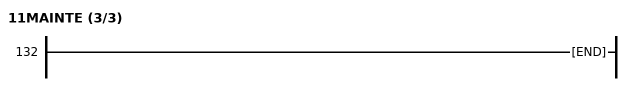
[picture p48: ladder of 11MAINTE, rungs at steps 132 to 132]
132   END
END_PROGRAM

PROGRAM 12ALARM1
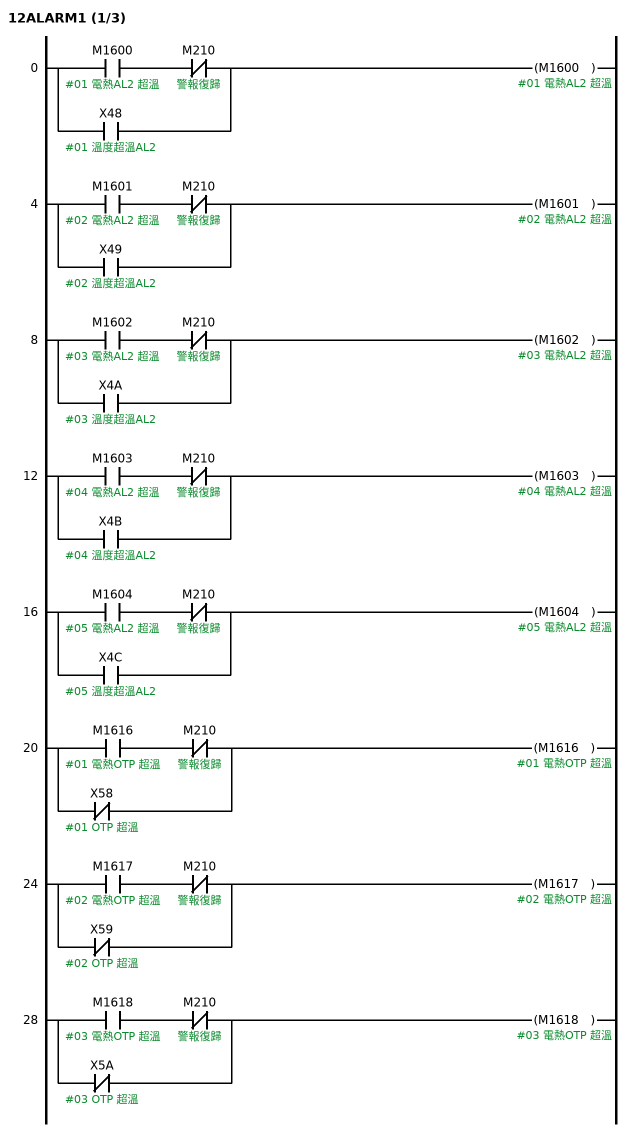
0     LD      M1600  ; #01 電熱AL2 超溫
      ANI     M210  ; 警報復歸
      OR      X48  ; #01 溫度超溫AL2
      OUT     M1600  ; #01 電熱AL2 超溫
4     LD      M1601  ; #02 電熱AL2 超溫
      ANI     M210  ; 警報復歸
      OR      X49  ; #02 溫度超溫AL2
      OUT     M1601  ; #02 電熱AL2 超溫
8     LD      M1602  ; #03 電熱AL2 超溫
      ANI     M210  ; 警報復歸
      OR      X4A  ; #03 溫度超溫AL2
      OUT     M1602  ; #03 電熱AL2 超溫
12    LD      M1603  ; #04 電熱AL2 超溫
      ANI     M210  ; 警報復歸
      OR      X4B  ; #04 溫度超溫AL2
      OUT     M1603  ; #04 電熱AL2 超溫
16    LD      M1604  ; #05 電熱AL2 超溫
      ANI     M210  ; 警報復歸
      OR      X4C  ; #05 溫度超溫AL2
      OUT     M1604  ; #05 電熱AL2 超溫
20    LD      M1616  ; #01 電熱OTP 超溫
      ANI     M210  ; 警報復歸
      ORI     X58  ; #01 OTP 超溫
      OUT     M1616  ; #01 電熱OTP 超溫
24    LD      M1617  ; #02 電熱OTP 超溫
      ANI     M210  ; 警報復歸
      ORI     X59  ; #02 OTP 超溫
      OUT     M1617  ; #02 電熱OTP 超溫
28    LD      M1618  ; #03 電熱OTP 超溫
      ANI     M210  ; 警報復歸
      ORI     X5A  ; #03 OTP 超溫
      OUT     M1618  ; #03 電熱OTP 超溫
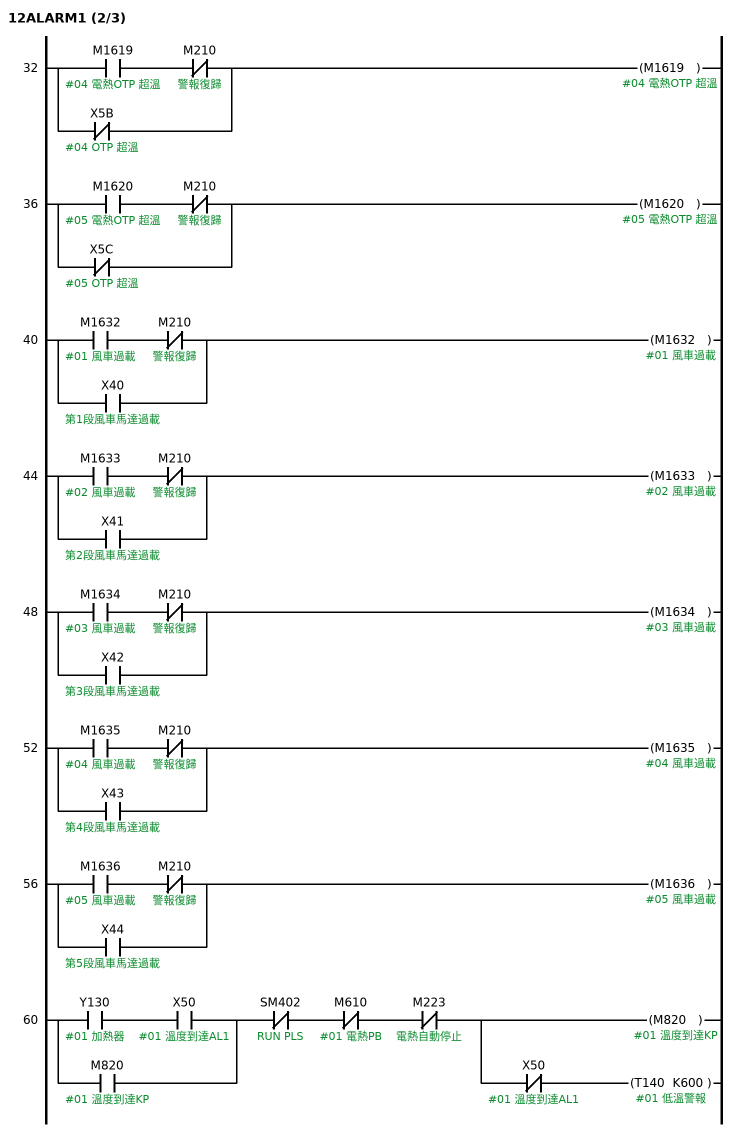
32    LD      M1619  ; #04 電熱OTP 超溫
      ANI     M210  ; 警報復歸
      ORI     X5B  ; #04 OTP 超溫
      OUT     M1619  ; #04 電熱OTP 超溫
36    LD      M1620  ; #05 電熱OTP 超溫
      ANI     M210  ; 警報復歸
      ORI     X5C  ; #05 OTP 超溫
      OUT     M1620  ; #05 電熱OTP 超溫
40    LD      M1632  ; #01 風車過載
      ANI     M210  ; 警報復歸
      OR      X40  ; 第1段風車馬達過載
      OUT     M1632  ; #01 風車過載
44    LD      M1633  ; #02 風車過載
      ANI     M210  ; 警報復歸
      OR      X41  ; 第2段風車馬達過載
      OUT     M1633  ; #02 風車過載
48    LD      M1634  ; #03 風車過載
      ANI     M210  ; 警報復歸
      OR      X42  ; 第3段風車馬達過載
      OUT     M1634  ; #03 風車過載
52    LD      M1635  ; #04 風車過載
      ANI     M210  ; 警報復歸
      OR      X43  ; 第4段風車馬達過載
      OUT     M1635  ; #04 風車過載
56    LD      M1636  ; #05 風車過載
      ANI     M210  ; 警報復歸
      OR      X44  ; 第5段風車馬達過載
      OUT     M1636  ; #05 風車過載
60    LD      Y130  ; #01 加熱器
      AND     X50  ; #01 溫度到達AL1
      OR      M820  ; #01 溫度到達KP
      ANI     SM402  ; RUN PLS
      ANI     M610  ; #01 電熱PB
      ANI     M223  ; 電熱自動停止
      OUT     M820  ; #01 溫度到達KP
      ANI     X50  ; #01 溫度到達AL1
      OUT     T140 K600  ; #01 低溫警報
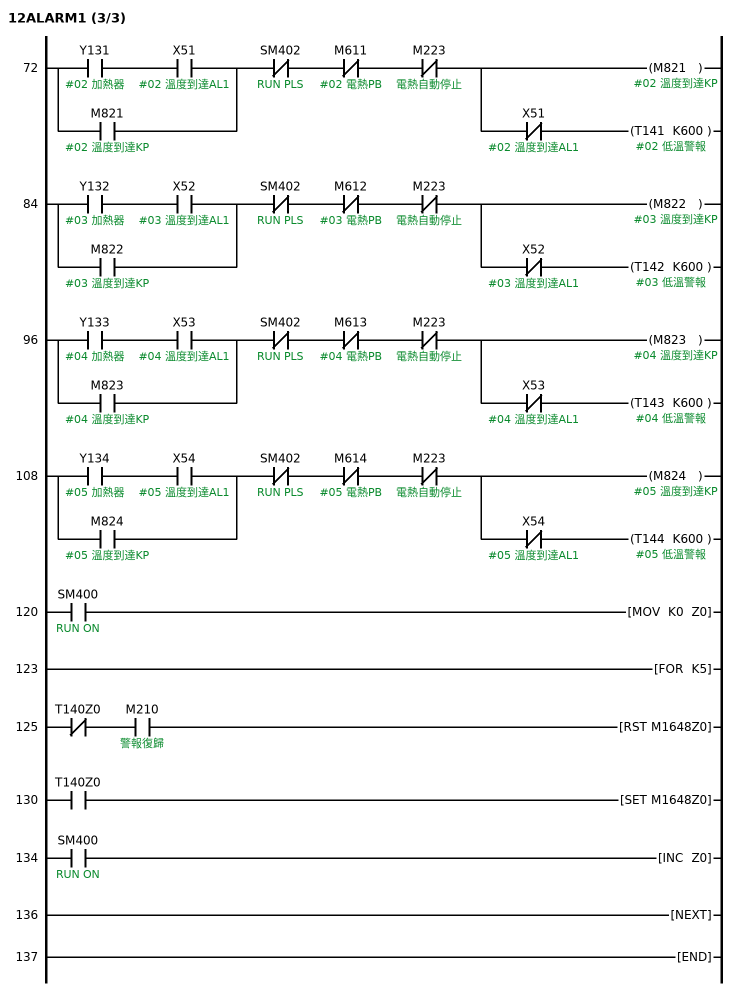
72    LD      Y131  ; #02 加熱器
      AND     X51  ; #02 溫度到達AL1
      OR      M821  ; #02 溫度到達KP
      ANI     SM402  ; RUN PLS
      ANI     M611  ; #02 電熱PB
      ANI     M223  ; 電熱自動停止
      OUT     M821  ; #02 溫度到達KP
      ANI     X51  ; #02 溫度到達AL1
      OUT     T141 K600  ; #02 低溫警報
84    LD      Y132  ; #03 加熱器
      AND     X52  ; #03 溫度到達AL1
      OR      M822  ; #03 溫度到達KP
      ANI     SM402  ; RUN PLS
      ANI     M612  ; #03 電熱PB
      ANI     M223  ; 電熱自動停止
      OUT     M822  ; #03 溫度到達KP
      ANI     X52  ; #03 溫度到達AL1
      OUT     T142 K600  ; #03 低溫警報
96    LD      Y133  ; #04 加熱器
      AND     X53  ; #04 溫度到達AL1
      OR      M823  ; #04 溫度到達KP
      ANI     SM402  ; RUN PLS
      ANI     M613  ; #04 電熱PB
      ANI     M223  ; 電熱自動停止
      OUT     M823  ; #04 溫度到達KP
      ANI     X53  ; #04 溫度到達AL1
      OUT     T143 K600  ; #04 低溫警報
108   LD      Y134  ; #05 加熱器
      AND     X54  ; #05 溫度到達AL1
      OR      M824  ; #05 溫度到達KP
      ANI     SM402  ; RUN PLS
      ANI     M614  ; #05 電熱PB
      ANI     M223  ; 電熱自動停止
      OUT     M824  ; #05 溫度到達KP
      ANI     X54  ; #05 溫度到達AL1
      OUT     T144 K600  ; #05 低溫警報
120   LD      SM400  ; RUN ON
      MOV     K0 Z0
123   FOR     K5
125   LDI     T140Z0
      AND     M210  ; 警報復歸
      RST     M1648Z0
130   LD      T140Z0
      SET     M1648Z0
134   LD      SM400  ; RUN ON
      INC     Z0
136   NEXT
137   END
END_PROGRAM

PROGRAM 13ALARM2
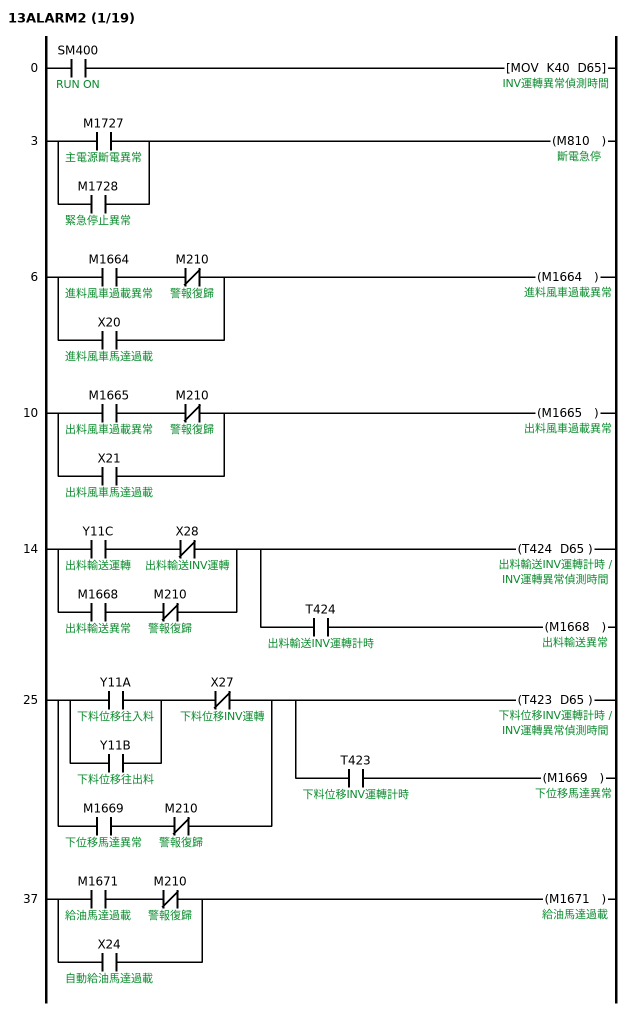
0     LD      SM400  ; RUN ON
      MOV     K40 D65  ; INV運轉異常偵測時間
3     LD      M1727  ; 主電源斷電異常
      OR      M1728  ; 緊急停止異常
      OUT     M810  ; 斷電急停
6     LD      M1664  ; 進料風車過載異常
      ANI     M210  ; 警報復歸
      OR      X20  ; 進料風車馬達過載
      OUT     M1664  ; 進料風車過載異常
10    LD      M1665  ; 出料風車過載異常
      ANI     M210  ; 警報復歸
      OR      X21  ; 出料風車馬達過載
      OUT     M1665  ; 出料風車過載異常
14    LD      Y11C  ; 出料輸送運轉
      ANI     X28  ; 出料輸送INV運轉
      LD      M1668  ; 出料輸送異常
      ANI     M210  ; 警報復歸
      ORB
      OUT     T424 D65  ; 出料輸送INV運轉計時 / INV運轉異常偵測時間
      AND     T424  ; 出料輸送INV運轉計時
      OUT     M1668  ; 出料輸送異常
25    LD      Y11A  ; 下料位移往入料
      OR      Y11B  ; 下料位移往出料
      ANI     X27  ; 下料位移INV運轉
      LD      M1669  ; 下位移馬達異常
      ANI     M210  ; 警報復歸
      ORB
      OUT     T423 D65  ; 下料位移INV運轉計時 / INV運轉異常偵測時間
      AND     T423  ; 下料位移INV運轉計時
      OUT     M1669  ; 下位移馬達異常
37    LD      M1671  ; 給油馬達過載
      ANI     M210  ; 警報復歸
      OR      X24  ; 自動給油馬達過載
      OUT     M1671  ; 給油馬達過載
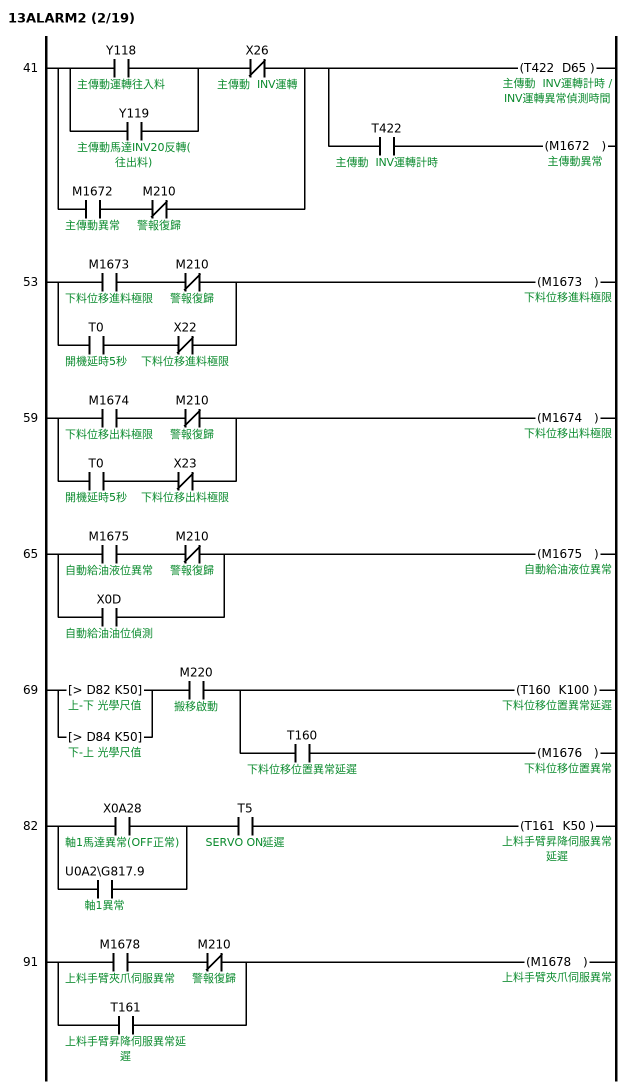
41    LD      Y118  ; 主傳動運轉往入料
      OR      Y119  ; 主傳動馬達INV20反轉(往出料)
      ANI     X26  ; 主傳動  INV運轉
      LD      M1672  ; 主傳動異常
      ANI     M210  ; 警報復歸
      ORB
      OUT     T422 D65  ; 主傳動  INV運轉計時 / INV運轉異常偵測時間
      AND     T422  ; 主傳動  INV運轉計時
      OUT     M1672  ; 主傳動異常
53    LD      M1673  ; 下料位移進料極限
      ANI     M210  ; 警報復歸
      LD      T0  ; 開機延時5秒
      ANI     X22  ; 下料位移進料極限
      ORB
      OUT     M1673  ; 下料位移進料極限
59    LD      M1674  ; 下料位移出料極限
      ANI     M210  ; 警報復歸
      LD      T0  ; 開機延時5秒
      ANI     X23  ; 下料位移出料極限
      ORB
      OUT     M1674  ; 下料位移出料極限
65    LD      M1675  ; 自動給油液位異常
      ANI     M210  ; 警報復歸
      OR      X0D  ; 自動給油油位偵測
      OUT     M1675  ; 自動給油液位異常
69    LD>     D82 K50  ; 上-下 光學尺值
      OR>     D84 K50  ; 下-上 光學尺值
      AND     M220  ; 搬移啟動
      OUT     T160 K100  ; 下料位移位置異常延遲
      AND     T160  ; 下料位移位置異常延遲
      OUT     M1676  ; 下料位移位置異常
82    LD      X0A28  ; 軸1馬達異常(OFF正常)
      OR      U0A2\G817.9  ; 軸1異常
      AND     T5  ; SERVO ON延遲
      OUT     T161 K50  ; 上料手臂昇降伺服異常延遲
91    LD      M1678  ; 上料手臂夾爪伺服異常
      ANI     M210  ; 警報復歸
      OR      T161  ; 上料手臂昇降伺服異常延遲
      OUT     M1678  ; 上料手臂夾爪伺服異常
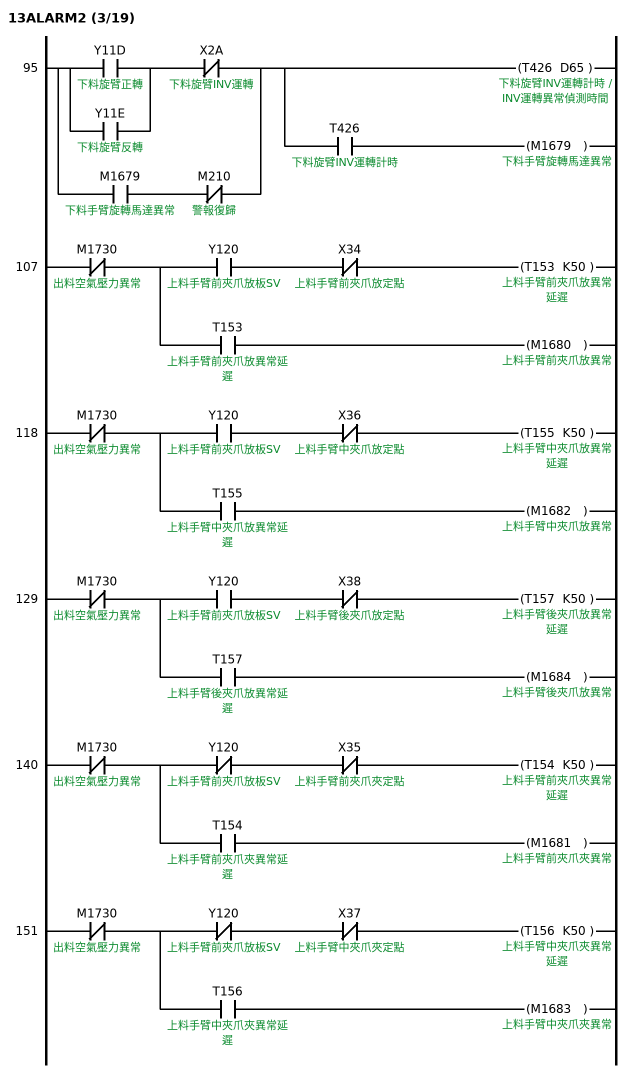
95    LD      Y11D  ; 下料旋臂正轉
      OR      Y11E  ; 下料旋臂反轉
      ANI     X2A  ; 下料旋臂INV運轉
      LD      M1679  ; 下料手臂旋轉馬達異常
      ANI     M210  ; 警報復歸
      ORB
      OUT     T426 D65  ; 下料旋臂INV運轉計時 / INV運轉異常偵測時間
      AND     T426  ; 下料旋臂INV運轉計時
      OUT     M1679  ; 下料手臂旋轉馬達異常
107   LDI     M1730  ; 出料空氣壓力異常
      MPS
      AND     Y120  ; 上料手臂前夾爪放板SV
      ANI     X34  ; 上料手臂前夾爪放定點
      OUT     T153 K50  ; 上料手臂前夾爪放異常延遲
      MPP
      AND     T153  ; 上料手臂前夾爪放異常延遲
      OUT     M1680  ; 上料手臂前夾爪放異常
118   LDI     M1730  ; 出料空氣壓力異常
      MPS
      AND     Y120  ; 上料手臂前夾爪放板SV
      ANI     X36  ; 上料手臂中夾爪放定點
      OUT     T155 K50  ; 上料手臂中夾爪放異常延遲
      MPP
      AND     T155  ; 上料手臂中夾爪放異常延遲
      OUT     M1682  ; 上料手臂中夾爪放異常
129   LDI     M1730  ; 出料空氣壓力異常
      MPS
      AND     Y120  ; 上料手臂前夾爪放板SV
      ANI     X38  ; 上料手臂後夾爪放定點
      OUT     T157 K50  ; 上料手臂後夾爪放異常延遲
      MPP
      AND     T157  ; 上料手臂後夾爪放異常延遲
      OUT     M1684  ; 上料手臂後夾爪放異常
140   LDI     M1730  ; 出料空氣壓力異常
      MPS
      ANI     Y120  ; 上料手臂前夾爪放板SV
      ANI     X35  ; 上料手臂前夾爪夾定點
      OUT     T154 K50  ; 上料手臂前夾爪夾異常延遲
      MPP
      AND     T154  ; 上料手臂前夾爪夾異常延遲
      OUT     M1681  ; 上料手臂前夾爪夾異常
151   LDI     M1730  ; 出料空氣壓力異常
      MPS
      ANI     Y120  ; 上料手臂前夾爪放板SV
      ANI     X37  ; 上料手臂中夾爪夾定點
      OUT     T156 K50  ; 上料手臂中夾爪夾異常延遲
      MPP
      AND     T156  ; 上料手臂中夾爪夾異常延遲
      OUT     M1683  ; 上料手臂中夾爪夾異常
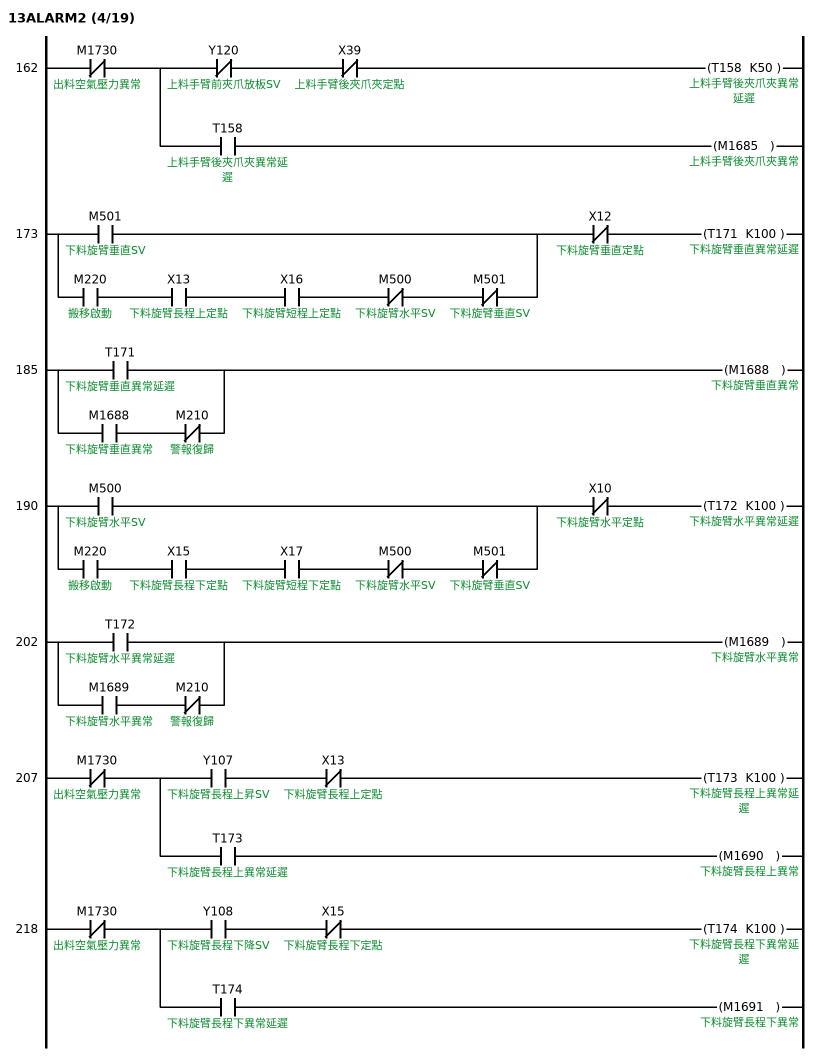
162   LDI     M1730  ; 出料空氣壓力異常
      MPS
      ANI     Y120  ; 上料手臂前夾爪放板SV
      ANI     X39  ; 上料手臂後夾爪夾定點
      OUT     T158 K50  ; 上料手臂後夾爪夾異常延遲
      MPP
      AND     T158  ; 上料手臂後夾爪夾異常延遲
      OUT     M1685  ; 上料手臂後夾爪夾異常
173   LD      M501  ; 下料旋臂垂直SV
      LD      M220  ; 搬移啟動
      AND     X13  ; 下料旋臂長程上定點
      AND     X16  ; 下料旋臂短程上定點
      ANI     M500  ; 下料旋臂水平SV
      ANI     M501  ; 下料旋臂垂直SV
      ORB
      ANI     X12  ; 下料旋臂垂直定點
      OUT     T171 K100  ; 下料旋臂垂直異常延遲
185   LD      T171  ; 下料旋臂垂直異常延遲
      LD      M1688  ; 下料旋臂垂直異常
      ANI     M210  ; 警報復歸
      ORB
      OUT     M1688  ; 下料旋臂垂直異常
190   LD      M500  ; 下料旋臂水平SV
      LD      M220  ; 搬移啟動
      AND     X15  ; 下料旋臂長程下定點
      AND     X17  ; 下料旋臂短程下定點
      ANI     M500  ; 下料旋臂水平SV
      ANI     M501  ; 下料旋臂垂直SV
      ORB
      ANI     X10  ; 下料旋臂水平定點
      OUT     T172 K100  ; 下料旋臂水平異常延遲
202   LD      T172  ; 下料旋臂水平異常延遲
      LD      M1689  ; 下料旋臂水平異常
      ANI     M210  ; 警報復歸
      ORB
      OUT     M1689  ; 下料旋臂水平異常
207   LDI     M1730  ; 出料空氣壓力異常
      MPS
      AND     Y107  ; 下料旋臂長程上昇SV
      ANI     X13  ; 下料旋臂長程上定點
      OUT     T173 K100  ; 下料旋臂長程上異常延遲
      MPP
      AND     T173  ; 下料旋臂長程上異常延遲
      OUT     M1690  ; 下料旋臂長程上異常
218   LDI     M1730  ; 出料空氣壓力異常
      MPS
      AND     Y108  ; 下料旋臂長程下降SV
      ANI     X15  ; 下料旋臂長程下定點
      OUT     T174 K100  ; 下料旋臂長程下異常延遲
      MPP
      AND     T174  ; 下料旋臂長程下異常延遲
      OUT     M1691  ; 下料旋臂長程下異常
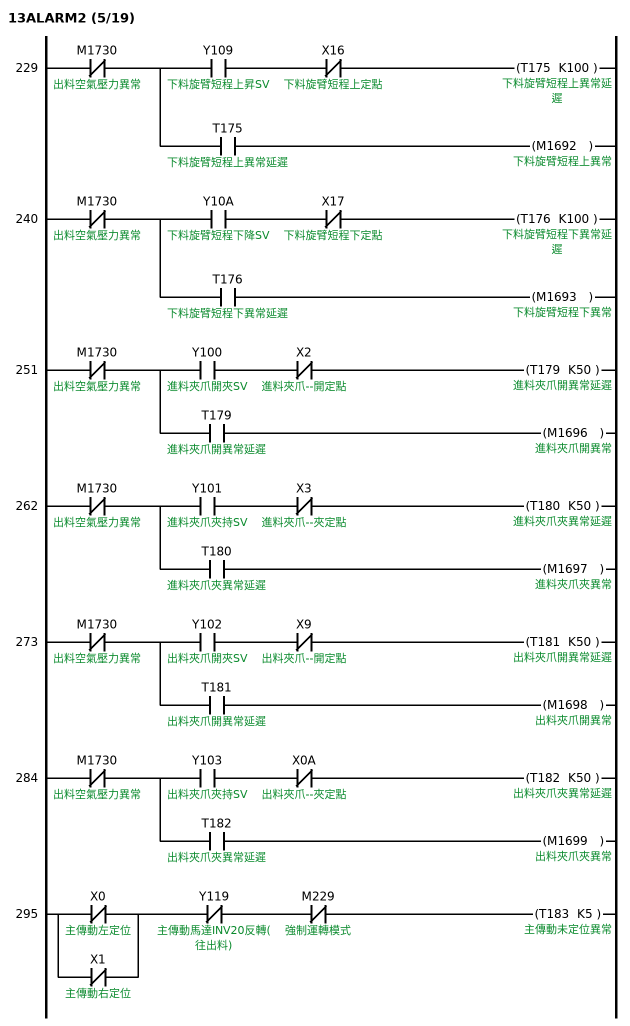
229   LDI     M1730  ; 出料空氣壓力異常
      MPS
      AND     Y109  ; 下料旋臂短程上昇SV
      ANI     X16  ; 下料旋臂短程上定點
      OUT     T175 K100  ; 下料旋臂短程上異常延遲
      MPP
      AND     T175  ; 下料旋臂短程上異常延遲
      OUT     M1692  ; 下料旋臂短程上異常
240   LDI     M1730  ; 出料空氣壓力異常
      MPS
      AND     Y10A  ; 下料旋臂短程下降SV
      ANI     X17  ; 下料旋臂短程下定點
      OUT     T176 K100  ; 下料旋臂短程下異常延遲
      MPP
      AND     T176  ; 下料旋臂短程下異常延遲
      OUT     M1693  ; 下料旋臂短程下異常
251   LDI     M1730  ; 出料空氣壓力異常
      MPS
      AND     Y100  ; 進料夾爪開夾SV
      ANI     X2  ; 進料夾爪--開定點
      OUT     T179 K50  ; 進料夾爪開異常延遲
      MPP
      AND     T179  ; 進料夾爪開異常延遲
      OUT     M1696  ; 進料夾爪開異常
262   LDI     M1730  ; 出料空氣壓力異常
      MPS
      AND     Y101  ; 進料夾爪夾持SV
      ANI     X3  ; 進料夾爪--夾定點
      OUT     T180 K50  ; 進料夾爪夾異常延遲
      MPP
      AND     T180  ; 進料夾爪夾異常延遲
      OUT     M1697  ; 進料夾爪夾異常
273   LDI     M1730  ; 出料空氣壓力異常
      MPS
      AND     Y102  ; 出料夾爪開夾SV
      ANI     X9  ; 出料夾爪--開定點
      OUT     T181 K50  ; 出料夾爪開異常延遲
      MPP
      AND     T181  ; 出料夾爪開異常延遲
      OUT     M1698  ; 出料夾爪開異常
284   LDI     M1730  ; 出料空氣壓力異常
      MPS
      AND     Y103  ; 出料夾爪夾持SV
      ANI     X0A  ; 出料夾爪--夾定點
      OUT     T182 K50  ; 出料夾爪夾異常延遲
      MPP
      AND     T182  ; 出料夾爪夾異常延遲
      OUT     M1699  ; 出料夾爪夾異常
295   LDI     X0  ; 主傳動左定位
      ORI     X1  ; 主傳動右定位
      ANI     Y119  ; 主傳動馬達INV20反轉(往出料)
      ANI     M229  ; 強制運轉模式
      OUT     T183 K5  ; 主傳動未定位異常
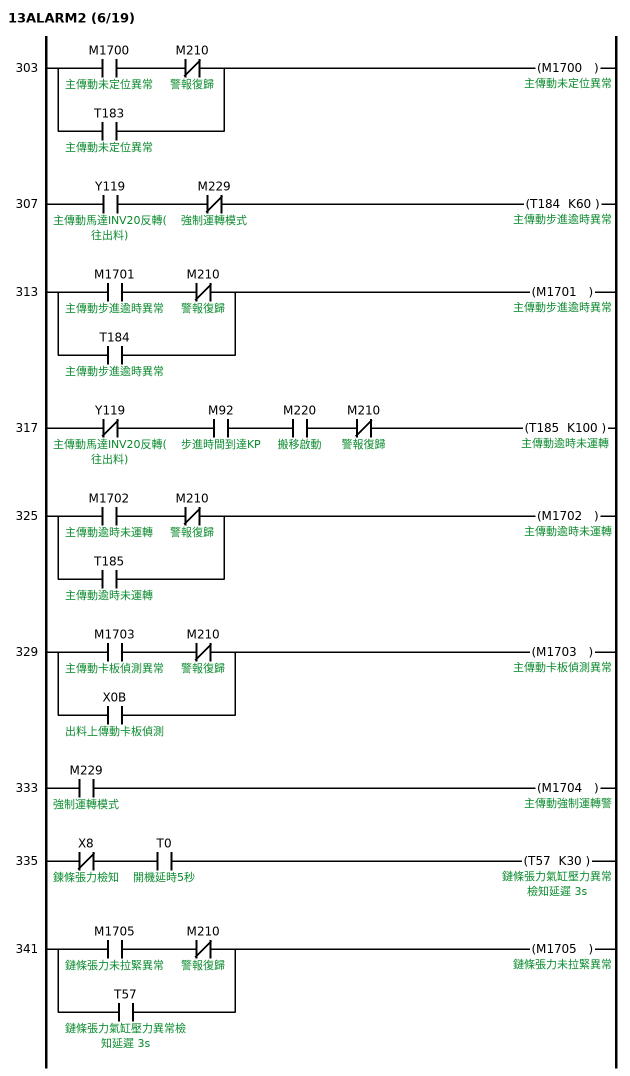
303   LD      M1700  ; 主傳動未定位異常
      ANI     M210  ; 警報復歸
      OR      T183  ; 主傳動未定位異常
      OUT     M1700  ; 主傳動未定位異常
307   LD      Y119  ; 主傳動馬達INV20反轉(往出料)
      ANI     M229  ; 強制運轉模式
      OUT     T184 K60  ; 主傳動步進逾時異常
313   LD      M1701  ; 主傳動步進逾時異常
      ANI     M210  ; 警報復歸
      OR      T184  ; 主傳動步進逾時異常
      OUT     M1701  ; 主傳動步進逾時異常
317   LDI     Y119  ; 主傳動馬達INV20反轉(往出料)
      AND     M92  ; 步進時間到達KP
      AND     M220  ; 搬移啟動
      ANI     M210  ; 警報復歸
      OUT     T185 K100  ; 主傳動逾時未運轉
325   LD      M1702  ; 主傳動逾時未運轉
      ANI     M210  ; 警報復歸
      OR      T185  ; 主傳動逾時未運轉
      OUT     M1702  ; 主傳動逾時未運轉
329   LD      M1703  ; 主傳動卡板偵測異常
      ANI     M210  ; 警報復歸
      OR      X0B  ; 出料上傳動卡板偵測
      OUT     M1703  ; 主傳動卡板偵測異常
333   LD      M229  ; 強制運轉模式
      OUT     M1704  ; 主傳動強制運轉警
335   LDI     X8  ; 鍊條張力檢知
      AND     T0  ; 開機延時5秒
      OUT     T57 K30  ; 鏈條張力氣缸壓力異常檢知延遲 3s
341   LD      M1705  ; 鏈條張力未拉緊異常
      ANI     M210  ; 警報復歸
      OR      T57  ; 鏈條張力氣缸壓力異常檢知延遲 3s
      OUT     M1705  ; 鏈條張力未拉緊異常
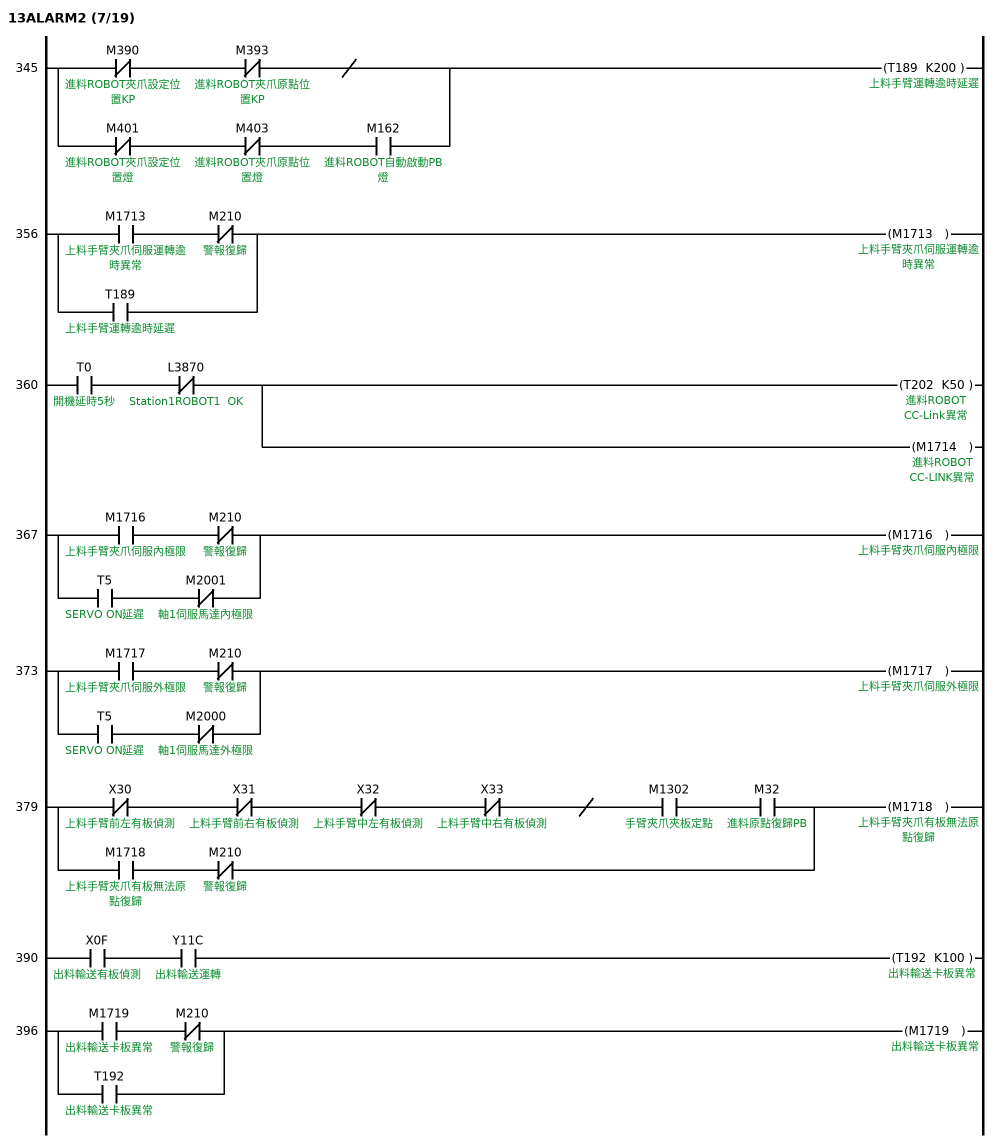
345   LDI     M390  ; 進料ROBOT夾爪設定位置KP
      ANI     M393  ; 進料ROBOT夾爪原點位置KP
      INV
      LDI     M401  ; 進料ROBOT夾爪設定位置燈
      ANI     M403  ; 進料ROBOT夾爪原點位置燈
      AND     M162  ; 進料ROBOT自動啟動PB燈
      ORB
      OUT     T189 K200  ; 上料手臂運轉逾時延遲
356   LD      M1713  ; 上料手臂夾爪伺服運轉逾時異常
      ANI     M210  ; 警報復歸
      OR      T189  ; 上料手臂運轉逾時延遲
      OUT     M1713  ; 上料手臂夾爪伺服運轉逾時異常
360   LD      T0  ; 開機延時5秒
      ANI     L3870  ; Station1ROBOT1  OK
      OUT     T202 K50  ; 進料ROBOT CC-Link異常
      OUT     M1714  ; 進料ROBOT CC-LINK異常
367   LD      M1716  ; 上料手臂夾爪伺服內極限
      ANI     M210  ; 警報復歸
      LD      T5  ; SERVO ON延遲
      ANI     M2001  ; 軸1伺服馬達內極限
      ORB
      OUT     M1716  ; 上料手臂夾爪伺服內極限
373   LD      M1717  ; 上料手臂夾爪伺服外極限
      ANI     M210  ; 警報復歸
      LD      T5  ; SERVO ON延遲
      ANI     M2000  ; 軸1伺服馬達外極限
      ORB
      OUT     M1717  ; 上料手臂夾爪伺服外極限
379   LDI     X30  ; 上料手臂前左有板偵測
      ANI     X31  ; 上料手臂前右有板偵測
      ANI     X32  ; 上料手臂中左有板偵測
      ANI     X33  ; 上料手臂中右有板偵測
      INV
      AND     M1302  ; 手臂夾爪夾板定點
      AND     M32  ; 進料原點復歸PB
      LD      M1718  ; 上料手臂夾爪有板無法原點復歸
      ANI     M210  ; 警報復歸
      ORB
      OUT     M1718  ; 上料手臂夾爪有板無法原點復歸
390   LD      X0F  ; 出料輸送有板偵測
      AND     Y11C  ; 出料輸送運轉
      OUT     T192 K100  ; 出料輸送卡板異常
396   LD      M1719  ; 出料輸送卡板異常
      ANI     M210  ; 警報復歸
      OR      T192  ; 出料輸送卡板異常
      OUT     M1719  ; 出料輸送卡板異常
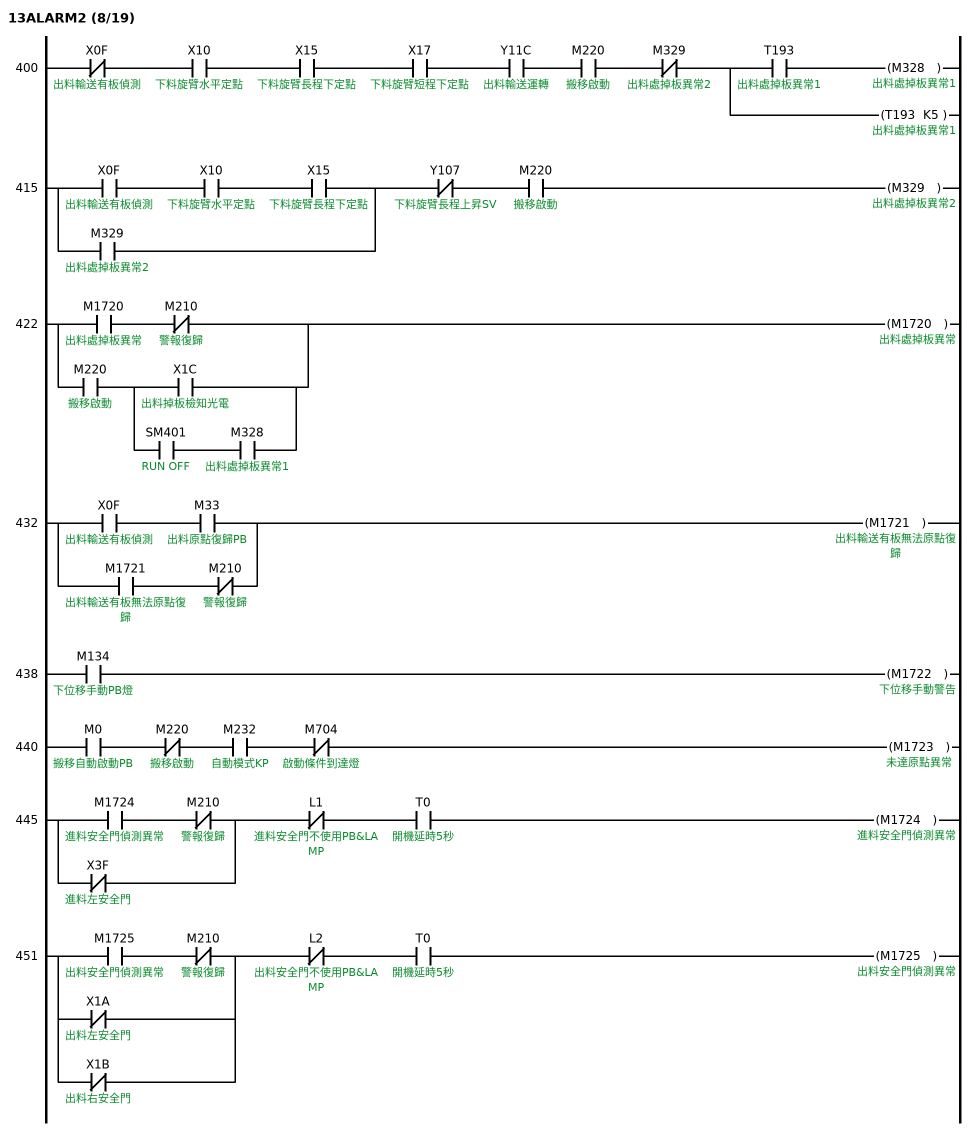
400   LDI     X0F  ; 出料輸送有板偵測
      AND     X10  ; 下料旋臂水平定點
      AND     X15  ; 下料旋臂長程下定點
      AND     X17  ; 下料旋臂短程下定點
      AND     Y11C  ; 出料輸送運轉
      AND     M220  ; 搬移啟動
      ANI     M329  ; 出料處掉板異常2
      MPS
      AND     T193  ; 出料處掉板異常1
      OUT     M328  ; 出料處掉板異常1
      MPP
      OUT     T193 K5  ; 出料處掉板異常1
415   LD      X0F  ; 出料輸送有板偵測
      AND     X10  ; 下料旋臂水平定點
      AND     X15  ; 下料旋臂長程下定點
      OR      M329  ; 出料處掉板異常2
      ANI     Y107  ; 下料旋臂長程上昇SV
      AND     M220  ; 搬移啟動
      OUT     M329  ; 出料處掉板異常2
422   LD      M1720  ; 出料處掉板異常
      ANI     M210  ; 警報復歸
      LD      M220  ; 搬移啟動
      LD      X1C  ; 出料掉板檢知光電
      LD      SM401  ; RUN OFF
      AND     M328  ; 出料處掉板異常1
      ORB
      ANB
      ORB
      OUT     M1720  ; 出料處掉板異常
432   LD      X0F  ; 出料輸送有板偵測
      AND     M33  ; 出料原點復歸PB
      LD      M1721  ; 出料輸送有板無法原點復歸
      ANI     M210  ; 警報復歸
      ORB
      OUT     M1721  ; 出料輸送有板無法原點復歸
438   LD      M134  ; 下位移手動PB燈
      OUT     M1722  ; 下位移手動警告
440   LD      M0  ; 搬移自動啟動PB
      ANI     M220  ; 搬移啟動
      AND     M232  ; 自動模式KP
      ANI     M704  ; 啟動條件到達燈
      OUT     M1723  ; 未達原點異常
445   LD      M1724  ; 進料安全門偵測異常
      ANI     M210  ; 警報復歸
      ORI     X3F  ; 進料左安全門
      ANI     L1  ; 進料安全門不使用PB&LAMP
      AND     T0  ; 開機延時5秒
      OUT     M1724  ; 進料安全門偵測異常
451   LD      M1725  ; 出料安全門偵測異常
      ANI     M210  ; 警報復歸
      ORI     X1A  ; 出料左安全門
      ORI     X1B  ; 出料右安全門
      ANI     L2  ; 出料安全門不使用PB&LAMP
      AND     T0  ; 開機延時5秒
      OUT     M1725  ; 出料安全門偵測異常
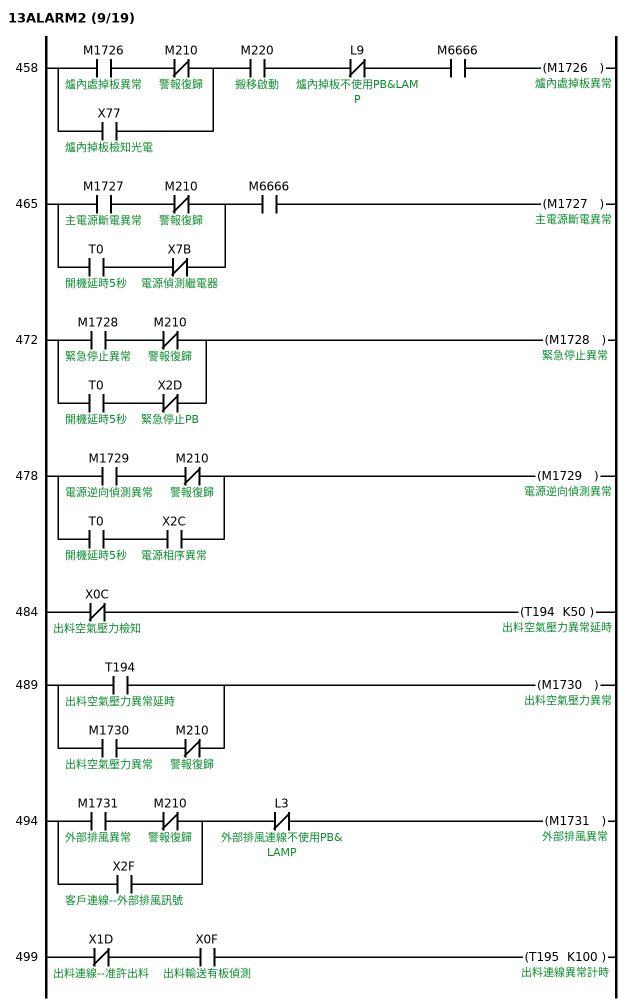
458   LD      M1726  ; 爐內處掉板異常
      ANI     M210  ; 警報復歸
      OR      X77  ; 爐內掉板檢知光電
      AND     M220  ; 搬移啟動
      ANI     L9  ; 爐內掉板不使用PB&LAMP
      AND     M6666
      OUT     M1726  ; 爐內處掉板異常
465   LD      M1727  ; 主電源斷電異常
      ANI     M210  ; 警報復歸
      LD      T0  ; 開機延時5秒
      ANI     X7B  ; 電源偵測繼電器
      ORB
      AND     M6666
      OUT     M1727  ; 主電源斷電異常
472   LD      M1728  ; 緊急停止異常
      ANI     M210  ; 警報復歸
      LD      T0  ; 開機延時5秒
      ANI     X2D  ; 緊急停止PB
      ORB
      OUT     M1728  ; 緊急停止異常
478   LD      M1729  ; 電源逆向偵測異常
      ANI     M210  ; 警報復歸
      LD      T0  ; 開機延時5秒
      AND     X2C  ; 電源相序異常
      ORB
      OUT     M1729  ; 電源逆向偵測異常
484   LDI     X0C  ; 出料空氣壓力檢知
      OUT     T194 K50  ; 出料空氣壓力異常延時
489   LD      T194  ; 出料空氣壓力異常延時
      LD      M1730  ; 出料空氣壓力異常
      ANI     M210  ; 警報復歸
      ORB
      OUT     M1730  ; 出料空氣壓力異常
494   LD      M1731  ; 外部排風異常
      ANI     M210  ; 警報復歸
      OR      X2F  ; 客戶連線--外部排風訊號
      ANI     L3  ; 外部排風連線不使用PB&LAMP
      OUT     M1731  ; 外部排風異常
499   LDI     X1D  ; 出料連線--准許出料
      AND     X0F  ; 出料輸送有板偵測
      OUT     T195 K100  ; 出料連線異常計時
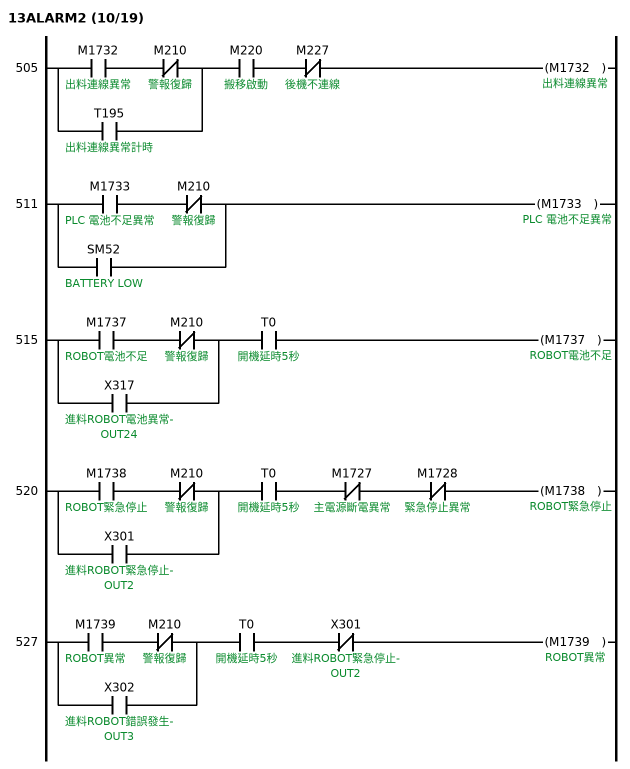
505   LD      M1732  ; 出料連線異常
      ANI     M210  ; 警報復歸
      OR      T195  ; 出料連線異常計時
      AND     M220  ; 搬移啟動
      ANI     M227  ; 後機不連線
      OUT     M1732  ; 出料連線異常
511   LD      M1733  ; PLC 電池不足異常
      ANI     M210  ; 警報復歸
      OR      SM52  ; BATTERY LOW
      OUT     M1733  ; PLC 電池不足異常
515   LD      M1737  ; ROBOT電池不足
      ANI     M210  ; 警報復歸
      OR      X317  ; 進料ROBOT電池異常-OUT24
      AND     T0  ; 開機延時5秒
      OUT     M1737  ; ROBOT電池不足
520   LD      M1738  ; ROBOT緊急停止
      ANI     M210  ; 警報復歸
      OR      X301  ; 進料ROBOT緊急停止-OUT2
      AND     T0  ; 開機延時5秒
      ANI     M1727  ; 主電源斷電異常
      ANI     M1728  ; 緊急停止異常
      OUT     M1738  ; ROBOT緊急停止
527   LD      M1739  ; ROBOT異常
      ANI     M210  ; 警報復歸
      OR      X302  ; 進料ROBOT錯誤發生-OUT3
      AND     T0  ; 開機延時5秒
      ANI     X301  ; 進料ROBOT緊急停止-OUT2
      OUT     M1739  ; ROBOT異常
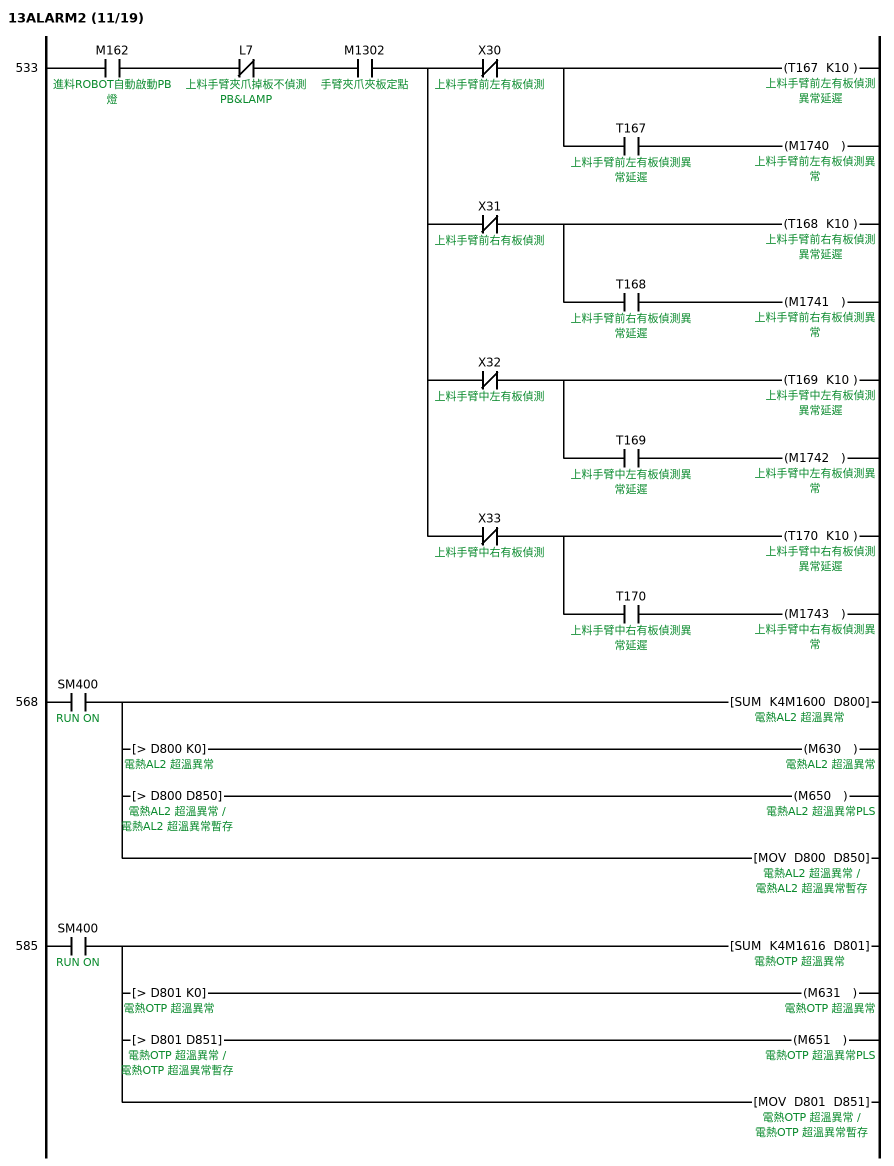
533   LD      M162  ; 進料ROBOT自動啟動PB燈
      ANI     L7  ; 上料手臂夾爪掉板不偵測PB&LAMP
      AND     M1302  ; 手臂夾爪夾板定點
      MPS
      ANI     X30  ; 上料手臂前左有板偵測
      OUT     T167 K10  ; 上料手臂前左有板偵測異常延遲
      AND     T167  ; 上料手臂前左有板偵測異常延遲
      OUT     M1740  ; 上料手臂前左有板偵測異常
      MRD
      ANI     X31  ; 上料手臂前右有板偵測
      OUT     T168 K10  ; 上料手臂前右有板偵測異常延遲
      AND     T168  ; 上料手臂前右有板偵測異常延遲
      OUT     M1741  ; 上料手臂前右有板偵測異常
      MRD
      ANI     X32  ; 上料手臂中左有板偵測
      OUT     T169 K10  ; 上料手臂中左有板偵測異常延遲
      AND     T169  ; 上料手臂中左有板偵測異常延遲
      OUT     M1742  ; 上料手臂中左有板偵測異常
      MPP
      ANI     X33  ; 上料手臂中右有板偵測
      OUT     T170 K10  ; 上料手臂中右有板偵測異常延遲
      AND     T170  ; 上料手臂中右有板偵測異常延遲
      OUT     M1743  ; 上料手臂中右有板偵測異常
568   LD      SM400  ; RUN ON
      SUM     K4M1600 D800  ; #01 電熱AL2 超溫 / 電熱AL2 超溫異常
      MPS
      AND>    D800 K0  ; 電熱AL2 超溫異常
      OUT     M630  ; 電熱AL2 超溫異常
      MRD
      AND>    D800 D850  ; 電熱AL2 超溫異常 / 電熱AL2 超溫異常暫存
      OUT     M650  ; 電熱AL2 超溫異常PLS
      MPP
      MOV     D800 D850
585   LD      SM400  ; RUN ON
      SUM     K4M1616 D801  ; #01 電熱OTP 超溫 / 電熱OTP 超溫異常
      MPS
      AND>    D801 K0  ; 電熱OTP 超溫異常
      OUT     M631  ; 電熱OTP 超溫異常
      MRD
      AND>    D801 D851  ; 電熱OTP 超溫異常 / 電熱OTP 超溫異常暫存
      OUT     M651  ; 電熱OTP 超溫異常PLS
      MPP
      MOV     D801 D851
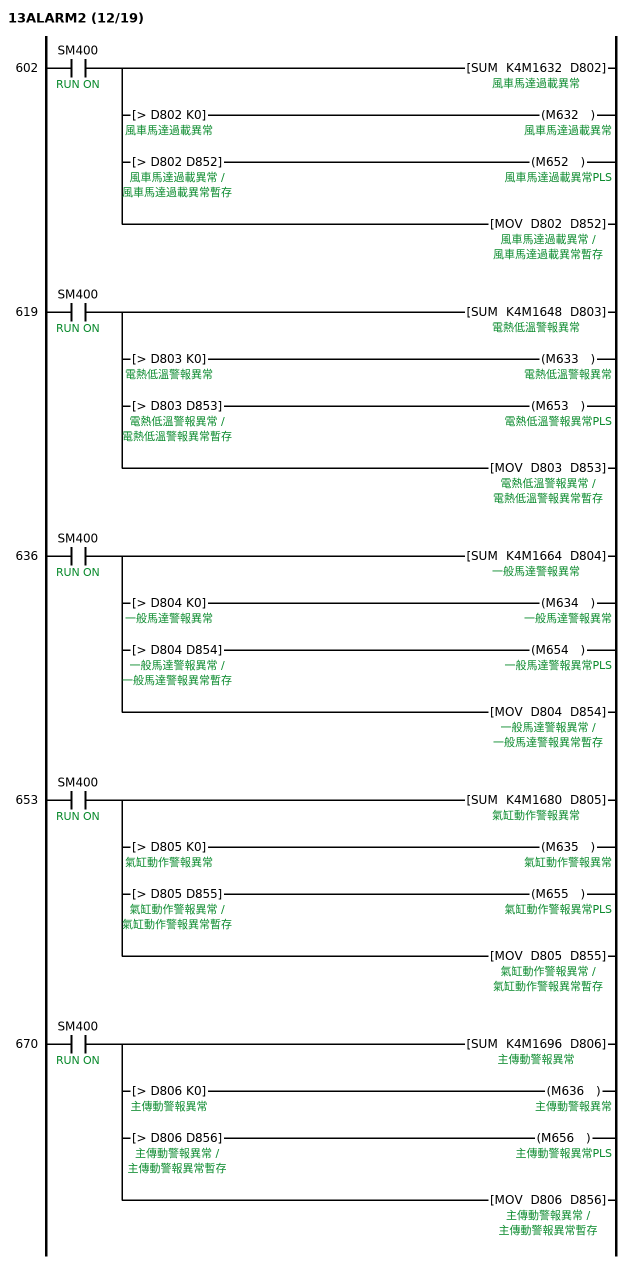
602   LD      SM400  ; RUN ON
      SUM     K4M1632 D802  ; #01 風車過載 / 風車馬達過載異常
      MPS
      AND>    D802 K0  ; 風車馬達過載異常
      OUT     M632  ; 風車馬達過載異常
      MRD
      AND>    D802 D852  ; 風車馬達過載異常 / 風車馬達過載異常暫存
      OUT     M652  ; 風車馬達過載異常PLS
      MPP
      MOV     D802 D852
619   LD      SM400  ; RUN ON
      SUM     K4M1648 D803  ; #01 低溫警報 / 電熱低溫警報異常
      MPS
      AND>    D803 K0  ; 電熱低溫警報異常
      OUT     M633  ; 電熱低溫警報異常
      MRD
      AND>    D803 D853  ; 電熱低溫警報異常 / 電熱低溫警報異常暫存
      OUT     M653  ; 電熱低溫警報異常PLS
      MPP
      MOV     D803 D853
636   LD      SM400  ; RUN ON
      SUM     K4M1664 D804  ; 一般馬達警報異常
      MPS
      AND>    D804 K0  ; 一般馬達警報異常
      OUT     M634  ; 一般馬達警報異常
      MRD
      AND>    D804 D854  ; 一般馬達警報異常 / 一般馬達警報異常暫存
      OUT     M654  ; 一般馬達警報異常PLS
      MPP
      MOV     D804 D854
653   LD      SM400  ; RUN ON
      SUM     K4M1680 D805  ; 氣缸動作警報異常
      MPS
      AND>    D805 K0  ; 氣缸動作警報異常
      OUT     M635  ; 氣缸動作警報異常
      MRD
      AND>    D805 D855  ; 氣缸動作警報異常 / 氣缸動作警報異常暫存
      OUT     M655  ; 氣缸動作警報異常PLS
      MPP
      MOV     D805 D855
670   LD      SM400  ; RUN ON
      SUM     K4M1696 D806  ; 主傳動警報異常
      MPS
      AND>    D806 K0  ; 主傳動警報異常
      OUT     M636  ; 主傳動警報異常
      MRD
      AND>    D806 D856  ; 主傳動警報異常 / 主傳動警報異常暫存
      OUT     M656  ; 主傳動警報異常PLS
      MPP
      MOV     D806 D856
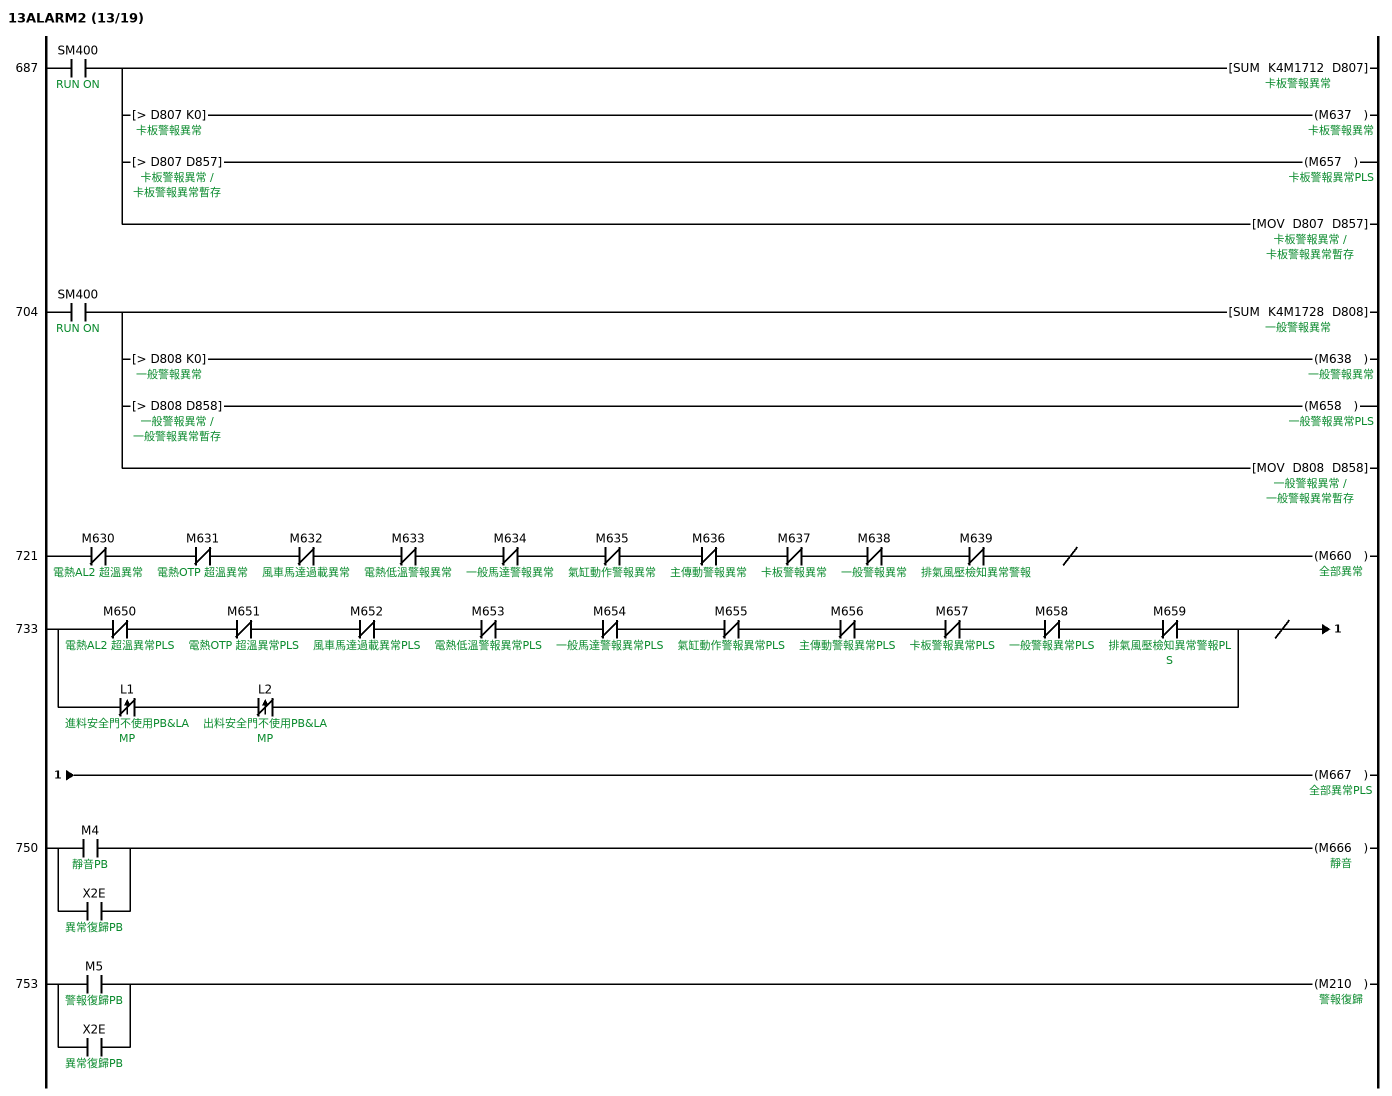
687   LD      SM400  ; RUN ON
      SUM     K4M1712 D807  ; 卡板警報異常
      MPS
      AND>    D807 K0  ; 卡板警報異常
      OUT     M637  ; 卡板警報異常
      MRD
      AND>    D807 D857  ; 卡板警報異常 / 卡板警報異常暫存
      OUT     M657  ; 卡板警報異常PLS
      MPP
      MOV     D807 D857
704   LD      SM400  ; RUN ON
      SUM     K4M1728 D808  ; 一般警報異常
      MPS
      AND>    D808 K0  ; 一般警報異常
      OUT     M638  ; 一般警報異常
      MRD
      AND>    D808 D858  ; 一般警報異常 / 一般警報異常暫存
      OUT     M658  ; 一般警報異常PLS
      MPP
      MOV     D808 D858
721   LDI     M630  ; 電熱AL2 超溫異常
      ANI     M631  ; 電熱OTP 超溫異常
      ANI     M632  ; 風車馬達過載異常
      ANI     M633  ; 電熱低溫警報異常
      ANI     M634  ; 一般馬達警報異常
      ANI     M635  ; 氣缸動作警報異常
      ANI     M636  ; 主傳動警報異常
      ANI     M637  ; 卡板警報異常
      ANI     M638  ; 一般警報異常
      ANI     M639  ; 排氣風壓檢知異常警報
      INV
      OUT     M660  ; 全部異常
733   LDI     M650  ; 電熱AL2 超溫異常PLS
      ANI     M651  ; 電熱OTP 超溫異常PLS
      ANI     M652  ; 風車馬達過載異常PLS
      ANI     M653  ; 電熱低溫警報異常PLS
      ANI     M654  ; 一般馬達警報異常PLS
      ANI     M655  ; 氣缸動作警報異常PLS
      ANI     M656  ; 主傳動警報異常PLS
      ANI     M657  ; 卡板警報異常PLS
      ANI     M658  ; 一般警報異常PLS
      ANI     M659  ; 排氣風壓檢知異常警報PLS
      LDPI    L1  ; 進料安全門不使用PB&LAMP
      ANDPI   L2  ; 出料安全門不使用PB&LAMP
      ORB
      INV
      OUT     M667  ; 全部異常PLS
750   LD      M4  ; 靜音PB
      OR      X2E  ; 異常復歸PB
      OUT     M666  ; 靜音
753   LD      M5  ; 警報復歸PB
      OR      X2E  ; 異常復歸PB
      OUT     M210  ; 警報復歸
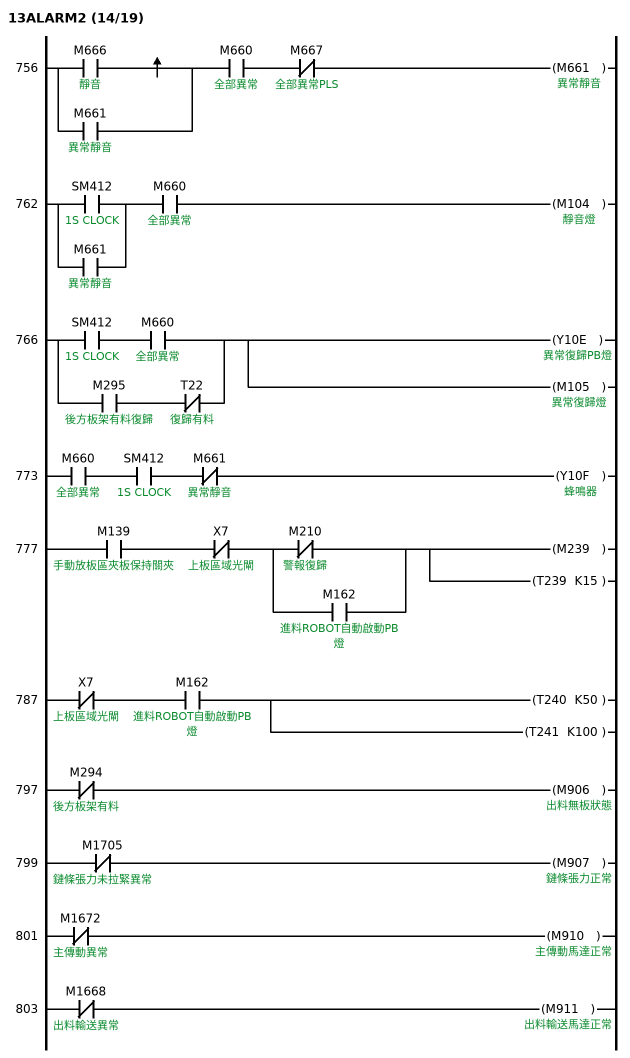
756   LD      M666  ; 靜音
      MEP
      OR      M661  ; 異常靜音
      AND     M660  ; 全部異常
      ANI     M667  ; 全部異常PLS
      OUT     M661  ; 異常靜音
762   LD      SM412  ; 1S CLOCK
      OR      M661  ; 異常靜音
      AND     M660  ; 全部異常
      OUT     M104  ; 靜音燈
766   LD      SM412  ; 1S CLOCK
      AND     M660  ; 全部異常
      LD      M295  ; 後方板架有料復歸
      ANI     T22  ; 復歸有料
      ORB
      OUT     Y10E  ; 異常復歸PB燈
      OUT     M105  ; 異常復歸燈
773   LD      M660  ; 全部異常
      AND     SM412  ; 1S CLOCK
      ANI     M661  ; 異常靜音
      OUT     Y10F  ; 蜂鳴器
777   LD      M139  ; 手動放板區夾板保持關夾
      ANI     X7  ; 上板區域光閘
      LDI     M210  ; 警報復歸
      OR      M162  ; 進料ROBOT自動啟動PB燈
      ANB
      OUT     M239
      OUT     T239 K15
787   LDI     X7  ; 上板區域光閘
      AND     M162  ; 進料ROBOT自動啟動PB燈
      OUT     T240 K50
      OUT     T241 K100
797   LDI     M294  ; 後方板架有料
      OUT     M906  ; 出料無板狀態
799   LDI     M1705  ; 鏈條張力未拉緊異常
      OUT     M907  ; 鏈條張力正常
801   LDI     M1672  ; 主傳動異常
      OUT     M910  ; 主傳動馬達正常
803   LDI     M1668  ; 出料輸送異常
      OUT     M911  ; 出料輸送馬達正常
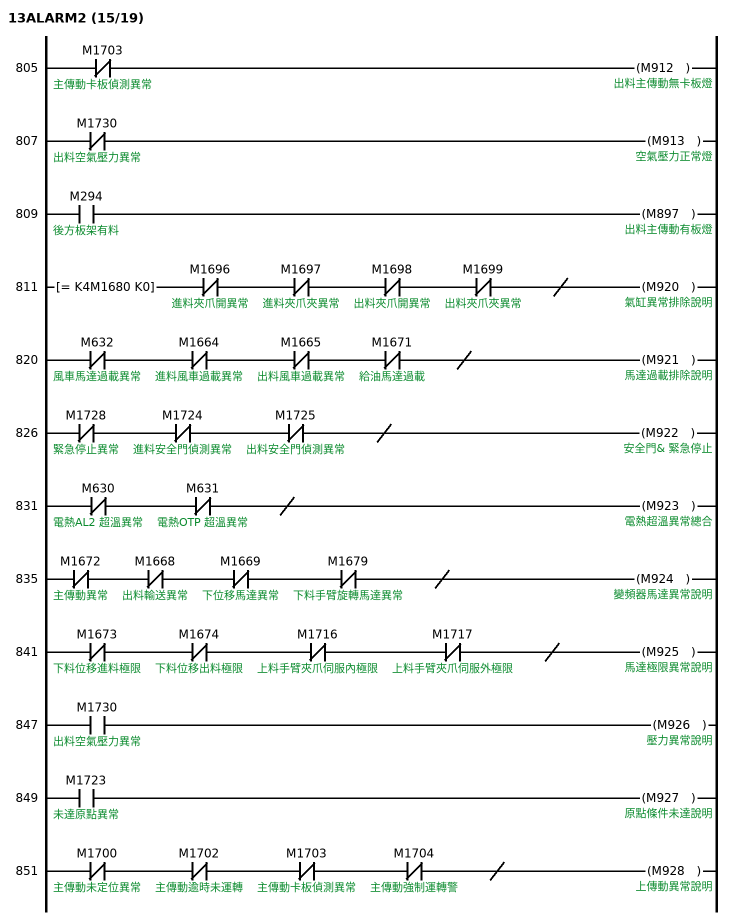
805   LDI     M1703  ; 主傳動卡板偵測異常
      OUT     M912  ; 出料主傳動無卡板燈
807   LDI     M1730  ; 出料空氣壓力異常
      OUT     M913  ; 空氣壓力正常燈
809   LD      M294  ; 後方板架有料
      OUT     M897  ; 出料主傳動有板燈
811   LD=     K4M1680 K0  ; 上料手臂前夾爪放異常
      ANI     M1696  ; 進料夾爪開異常
      ANI     M1697  ; 進料夾爪夾異常
      ANI     M1698  ; 出料夾爪開異常
      ANI     M1699  ; 出料夾爪夾異常
      INV
      OUT     M920  ; 氣缸異常排除說明
820   LDI     M632  ; 風車馬達過載異常
      ANI     M1664  ; 進料風車過載異常
      ANI     M1665  ; 出料風車過載異常
      ANI     M1671  ; 給油馬達過載
      INV
      OUT     M921  ; 馬達過載排除說明
826   LDI     M1728  ; 緊急停止異常
      ANI     M1724  ; 進料安全門偵測異常
      ANI     M1725  ; 出料安全門偵測異常
      INV
      OUT     M922  ; 安全門& 緊急停止
831   LDI     M630  ; 電熱AL2 超溫異常
      ANI     M631  ; 電熱OTP 超溫異常
      INV
      OUT     M923  ; 電熱超溫異常總合
835   LDI     M1672  ; 主傳動異常
      ANI     M1668  ; 出料輸送異常
      ANI     M1669  ; 下位移馬達異常
      ANI     M1679  ; 下料手臂旋轉馬達異常
      INV
      OUT     M924  ; 變頻器馬達異常說明
841   LDI     M1673  ; 下料位移進料極限
      ANI     M1674  ; 下料位移出料極限
      ANI     M1716  ; 上料手臂夾爪伺服內極限
      ANI     M1717  ; 上料手臂夾爪伺服外極限
      INV
      OUT     M925  ; 馬達極限異常說明
847   LD      M1730  ; 出料空氣壓力異常
      OUT     M926  ; 壓力異常說明
849   LD      M1723  ; 未達原點異常
      OUT     M927  ; 原點條件未達說明
851   LDI     M1700  ; 主傳動未定位異常
      ANI     M1702  ; 主傳動逾時未運轉
      ANI     M1703  ; 主傳動卡板偵測異常
      ANI     M1704  ; 主傳動強制運轉警
      INV
      OUT     M928  ; 上傳動異常說明
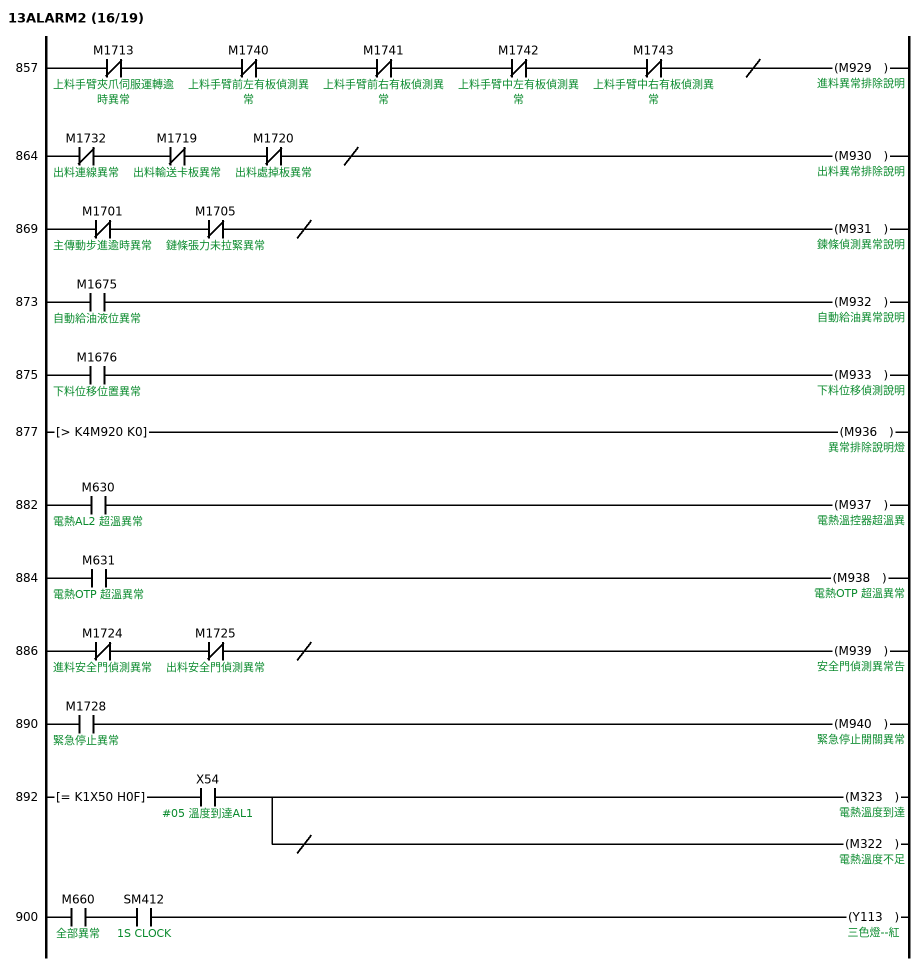
857   LDI     M1713  ; 上料手臂夾爪伺服運轉逾時異常
      ANI     M1740  ; 上料手臂前左有板偵測異常
      ANI     M1741  ; 上料手臂前右有板偵測異常
      ANI     M1742  ; 上料手臂中左有板偵測異常
      ANI     M1743  ; 上料手臂中右有板偵測異常
      INV
      OUT     M929  ; 進料異常排除說明
864   LDI     M1732  ; 出料連線異常
      ANI     M1719  ; 出料輸送卡板異常
      ANI     M1720  ; 出料處掉板異常
      INV
      OUT     M930  ; 出料異常排除說明
869   LDI     M1701  ; 主傳動步進逾時異常
      ANI     M1705  ; 鏈條張力未拉緊異常
      INV
      OUT     M931  ; 鍊條偵測異常說明
873   LD      M1675  ; 自動給油液位異常
      OUT     M932  ; 自動給油異常說明
875   LD      M1676  ; 下料位移位置異常
      OUT     M933  ; 下料位移偵測說明
877   LD>     K4M920 K0  ; 氣缸異常排除說明
      OUT     M936  ; 異常排除說明燈
882   LD      M630  ; 電熱AL2 超溫異常
      OUT     M937  ; 電熱溫控器超溫異
884   LD      M631  ; 電熱OTP 超溫異常
      OUT     M938  ; 電熱OTP 超溫異常
886   LDI     M1724  ; 進料安全門偵測異常
      ANI     M1725  ; 出料安全門偵測異常
      INV
      OUT     M939  ; 安全門偵測異常告
890   LD      M1728  ; 緊急停止異常
      OUT     M940  ; 緊急停止開關異常
892   LD=     K1X50 H0F  ; #01 溫度到達AL1
      AND     X54  ; #05 溫度到達AL1
      OUT     M323  ; 電熱溫度到達
      INV
      OUT     M322  ; 電熱溫度不足
900   LD      M660  ; 全部異常
      AND     SM412  ; 1S CLOCK
      OUT     Y113  ; 三色燈--紅
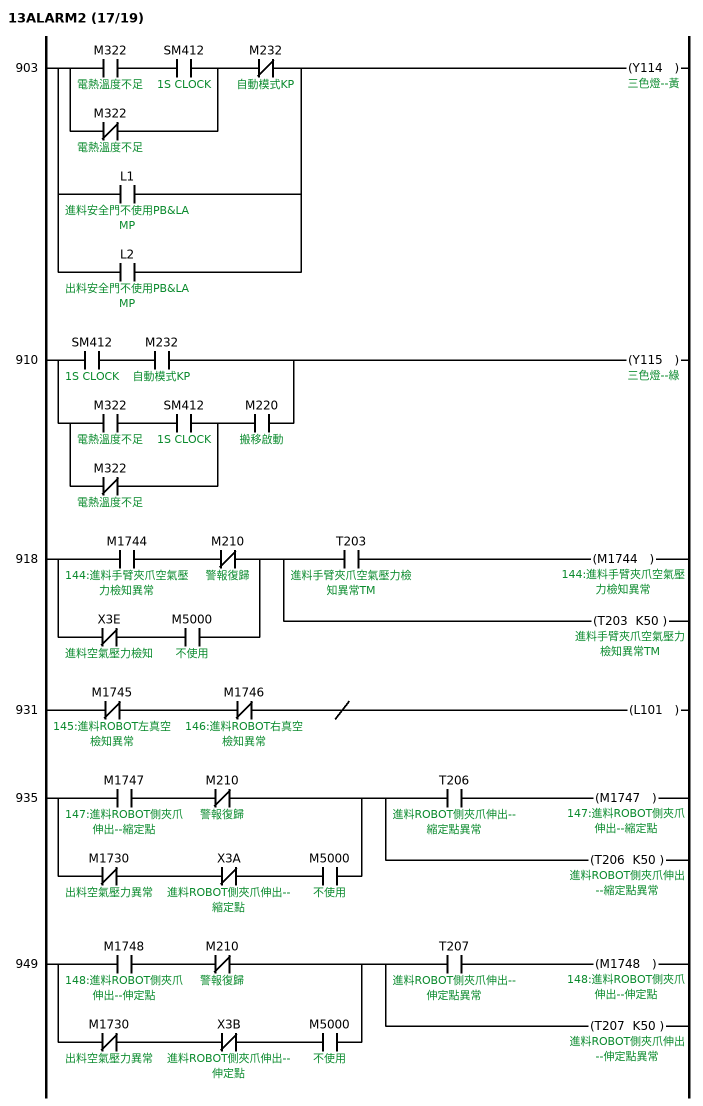
903   LD      M322  ; 電熱溫度不足
      AND     SM412  ; 1S CLOCK
      ORI     M322  ; 電熱溫度不足
      ANI     M232  ; 自動模式KP
      OR      L1  ; 進料安全門不使用PB&LAMP
      OR      L2  ; 出料安全門不使用PB&LAMP
      OUT     Y114  ; 三色燈--黃
910   LD      SM412  ; 1S CLOCK
      AND     M232  ; 自動模式KP
      LD      M322  ; 電熱溫度不足
      AND     SM412  ; 1S CLOCK
      ORI     M322  ; 電熱溫度不足
      AND     M220  ; 搬移啟動
      ORB
      OUT     Y115  ; 三色燈--綠
918   LD      M1744  ; 144:進料手臂夾爪空氣壓力檢知異常
      ANI     M210  ; 警報復歸
      LDI     X3E  ; 進料空氣壓力檢知
      AND     M5000  ; 不使用
      ORB
      MPS
      AND     T203  ; 進料手臂夾爪空氣壓力檢知異常TM
      OUT     M1744  ; 144:進料手臂夾爪空氣壓力檢知異常
      MPP
      OUT     T203 K50  ; 進料手臂夾爪空氣壓力檢知異常TM
931   LDI     M1745  ; 145:進料ROBOT左真空檢知異常
      ANI     M1746  ; 146:進料ROBOT右真空檢知異常
      INV
      OUT     L101
935   LD      M1747  ; 147:進料ROBOT側夾爪伸出--縮定點
      ANI     M210  ; 警報復歸
      LDI     M1730  ; 出料空氣壓力異常
      ANI     X3A  ; 進料ROBOT側夾爪伸出--縮定點
      AND     M5000  ; 不使用
      ORB
      MPS
      AND     T206  ; 進料ROBOT側夾爪伸出--縮定點異常
      OUT     M1747  ; 147:進料ROBOT側夾爪伸出--縮定點
      MPP
      OUT     T206 K50  ; 進料ROBOT側夾爪伸出--縮定點異常
949   LD      M1748  ; 148:進料ROBOT側夾爪伸出--伸定點
      ANI     M210  ; 警報復歸
      LDI     M1730  ; 出料空氣壓力異常
      ANI     X3B  ; 進料ROBOT側夾爪伸出--伸定點
      AND     M5000  ; 不使用
      ORB
      MPS
      AND     T207  ; 進料ROBOT側夾爪伸出--伸定點異常
      OUT     M1748  ; 148:進料ROBOT側夾爪伸出--伸定點
      MPP
      OUT     T207 K50  ; 進料ROBOT側夾爪伸出--伸定點異常
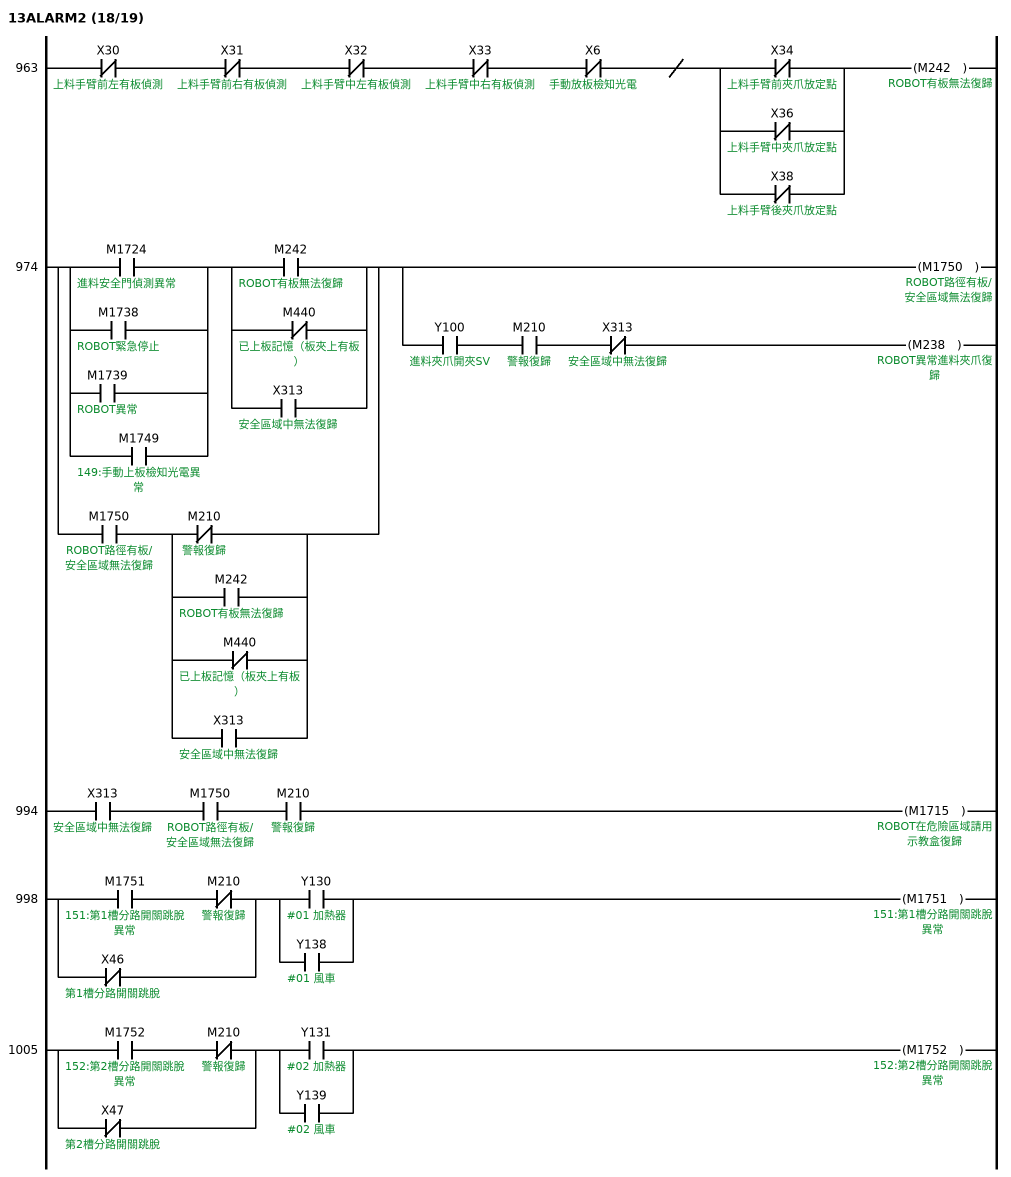
963   LDI     X30  ; 上料手臂前左有板偵測
      ANI     X31  ; 上料手臂前右有板偵測
      ANI     X32  ; 上料手臂中左有板偵測
      ANI     X33  ; 上料手臂中右有板偵測
      ANI     X6  ; 手動放板檢知光電
      INV
      LDI     X34  ; 上料手臂前夾爪放定點
      ORI     X36  ; 上料手臂中夾爪放定點
      ORI     X38  ; 上料手臂後夾爪放定點
      ANB
      OUT     M242  ; ROBOT有板無法復歸
974   LD      M1724  ; 進料安全門偵測異常
      OR      M1738  ; ROBOT緊急停止
      OR      M1739  ; ROBOT異常
      OR      M1749  ; 149:手動上板檢知光電異常
      LD      M242  ; ROBOT有板無法復歸
      ORI     M440  ; 已上板記憶（板夾上有板）
      OR      X313  ; 安全區域中無法復歸
      ANB
      LD      M1750  ; ROBOT路徑有板/安全區域無法復歸
      LDI     M210  ; 警報復歸
      OR      M242  ; ROBOT有板無法復歸
      ORI     M440  ; 已上板記憶（板夾上有板）
      OR      X313  ; 安全區域中無法復歸
      ANB
      ORB
      OUT     M1750  ; ROBOT路徑有板/安全區域無法復歸
      AND     Y100  ; 進料夾爪開夾SV
      AND     M210  ; 警報復歸
      ANI     X313  ; 安全區域中無法復歸
      OUT     M238  ; ROBOT異常進料夾爪復歸
994   LD      X313  ; 安全區域中無法復歸
      AND     M1750  ; ROBOT路徑有板/安全區域無法復歸
      AND     M210  ; 警報復歸
      OUT     M1715  ; ROBOT在危險區域請用示教盒復歸
998   LD      M1751  ; 151:第1槽分路開關跳脫異常
      ANI     M210  ; 警報復歸
      ORI     X46  ; 第1槽分路開關跳脫
      LD      Y130  ; #01 加熱器
      OR      Y138  ; #01 風車
      ANB
      OUT     M1751  ; 151:第1槽分路開關跳脫異常
1005  LD      M1752  ; 152:第2槽分路開關跳脫異常
      ANI     M210  ; 警報復歸
      ORI     X47  ; 第2槽分路開關跳脫
      LD      Y131  ; #02 加熱器
      OR      Y139  ; #02 風車
      ANB
      OUT     M1752  ; 152:第2槽分路開關跳脫異常
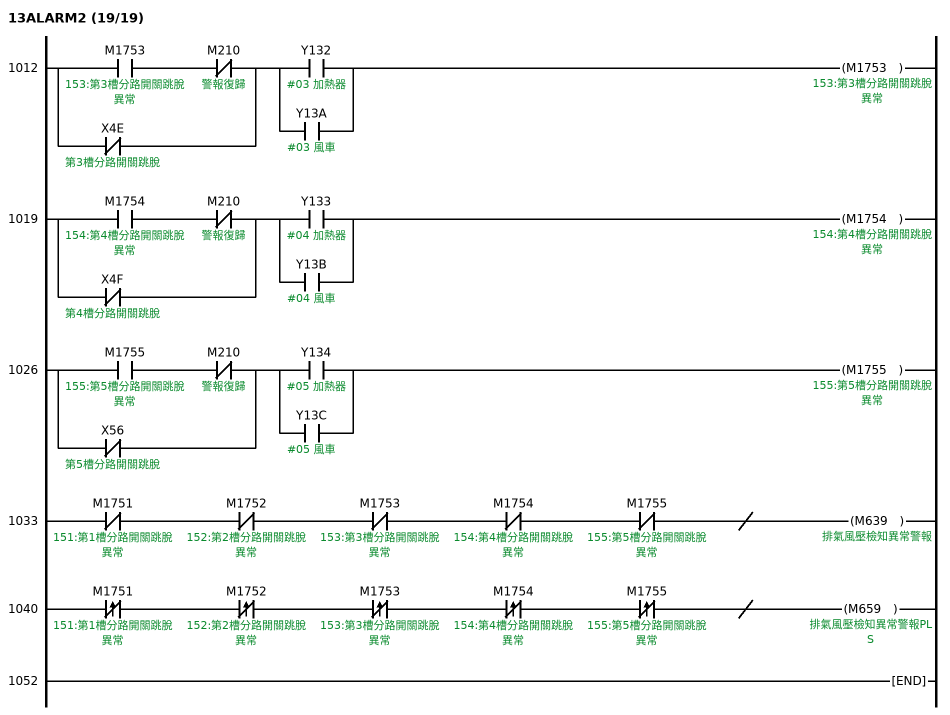
1012  LD      M1753  ; 153:第3槽分路開關跳脫異常
      ANI     M210  ; 警報復歸
      ORI     X4E  ; 第3槽分路開關跳脫
      LD      Y132  ; #03 加熱器
      OR      Y13A  ; #03 風車
      ANB
      OUT     M1753  ; 153:第3槽分路開關跳脫異常
1019  LD      M1754  ; 154:第4槽分路開關跳脫異常
      ANI     M210  ; 警報復歸
      ORI     X4F  ; 第4槽分路開關跳脫
      LD      Y133  ; #04 加熱器
      OR      Y13B  ; #04 風車
      ANB
      OUT     M1754  ; 154:第4槽分路開關跳脫異常
1026  LD      M1755  ; 155:第5槽分路開關跳脫異常
      ANI     M210  ; 警報復歸
      ORI     X56  ; 第5槽分路開關跳脫
      LD      Y134  ; #05 加熱器
      OR      Y13C  ; #05 風車
      ANB
      OUT     M1755  ; 155:第5槽分路開關跳脫異常
1033  LDI     M1751  ; 151:第1槽分路開關跳脫異常
      ANI     M1752  ; 152:第2槽分路開關跳脫異常
      ANI     M1753  ; 153:第3槽分路開關跳脫異常
      ANI     M1754  ; 154:第4槽分路開關跳脫異常
      ANI     M1755  ; 155:第5槽分路開關跳脫異常
      INV
      OUT     M639  ; 排氣風壓檢知異常警報
1040  LDPI    M1751  ; 151:第1槽分路開關跳脫異常
      ANDPI   M1752  ; 152:第2槽分路開關跳脫異常
      ANDPI   M1753  ; 153:第3槽分路開關跳脫異常
      ANDPI   M1754  ; 154:第4槽分路開關跳脫異常
      ANDPI   M1755  ; 155:第5槽分路開關跳脫異常
      INV
      OUT     M659  ; 排氣風壓檢知異常警報PLS
1052  END
END_PROGRAM

PROGRAM 14TIME
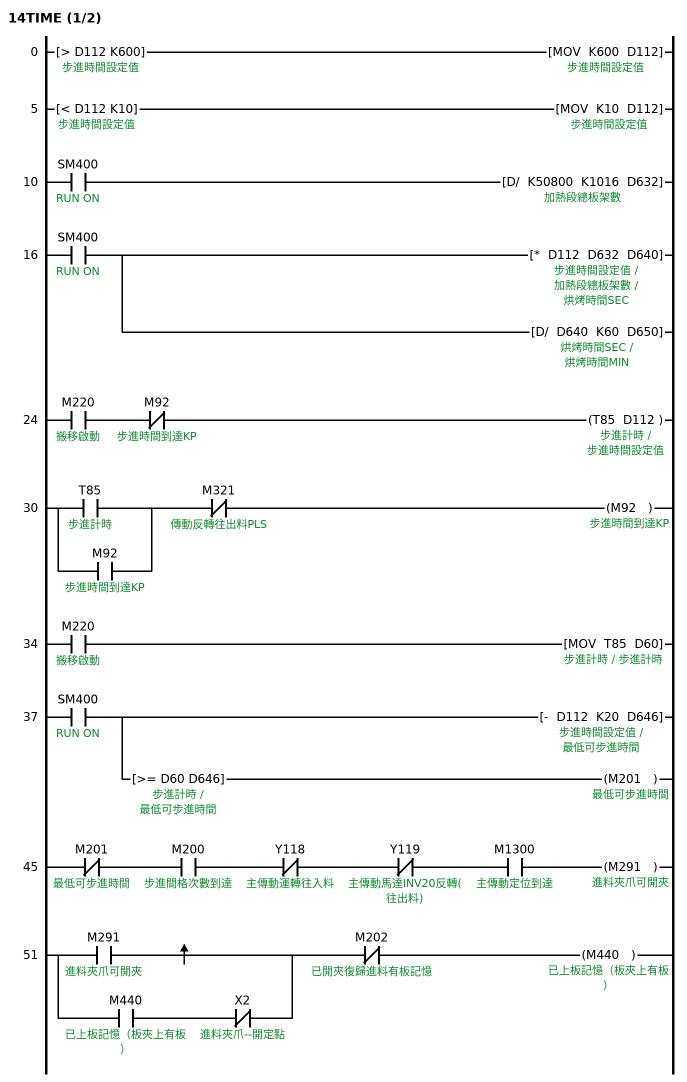
0     LD>     D112 K600  ; 步進時間設定值
      MOV     K600 D112
5     LD<     D112 K10  ; 步進時間設定值
      MOV     K10 D112
10    LD      SM400  ; RUN ON
      D/      K50800 K1016 D632  ; 加熱段總板架數
16    LD      SM400  ; RUN ON
      *       D112 D632 D640  ; 烘烤時間SEC
      D/      D640 K60 D650  ; 烘烤時間MIN
24    LD      M220  ; 搬移啟動
      ANI     M92  ; 步進時間到達KP
      OUT     T85 D112  ; 步進計時 / 步進時間設定值
30    LD      T85  ; 步進計時
      OR      M92  ; 步進時間到達KP
      ANI     M321  ; 傳動反轉往出料PLS
      OUT     M92  ; 步進時間到達KP
34    LD      M220  ; 搬移啟動
      MOV     T85 D60  ; 步進計時
37    LD      SM400  ; RUN ON
      -       D112 K20 D646  ; 最低可步進時間
      AND>=   D60 D646  ; 步進計時 / 最低可步進時間
      OUT     M201  ; 最低可步進時間
45    LDI     M201  ; 最低可步進時間
      AND     M200  ; 步進間格次數到達
      ANI     Y118  ; 主傳動運轉往入料
      ANI     Y119  ; 主傳動馬達INV20反轉(往出料)
      AND     M1300  ; 主傳動定位到達
      OUT     M291  ; 進料夾爪可開夾
51    LD      M291  ; 進料夾爪可開夾
      MEP
      LD      M440  ; 已上板記憶（板夾上有板）
      ANI     X2  ; 進料夾爪--開定點
      ORB
      ANI     M202  ; 已開夾復歸進料有板記憶
      OUT     M440  ; 已上板記憶（板夾上有板）
